LIN {X 0,Y 306.051,Z 523.216,A -85,B 0,C 180,E1 -15945.996,E2 -15945.996} C_VEL
LIN {X 0,Y 307.496,Z 515.084,A -85,B 0,C 180,E1 -15948.317,E2 -15948.317} C_VEL
LIN {X 0,Y 309.447,Z 505.284,A -85,B 0,C 180,E1 -15950.612,E2 -15950.612} C_VEL
LIN {X 0,Y 311.307,Z 495.226,A -85,B 0,C 180,E1 -15952.569,E2 -15952.569} C_VEL
LIN {X 0,Y 313.603,Z 483.236,A -85,B 0,C 180,E1 -15954.494,E2 -15954.494} C_VEL
LIN {X 0,Y 315.881,Z 471.244,A -85,B 0,C 180,E1 -15956.067,E2 -15956.067} C_VEL
LIN {X 0,Y 318.15,Z 458.217,A -85,B 0,C 180,E1 -15957.46,E2 -15957.46} C_VEL
LIN {X 0,Y 320.166,Z 444.237,A -85,B 0,C 180,E1 -15958.665,E2 -15958.665} C_VEL
LIN {X 0,Y 321.912,Z 430.188,A -85,B 0,C 180,E1 -15959.601,E2 -15959.601} C_VEL
LIN {X 0,Y 323.462,Z 414.88,A -85,B 0,C 180,E1 -15960.342,E2 -15960.342} C_VEL
LIN {X 0,Y 324.422,Z 399.961,A -85,B 0,C 180,E1 -15960.828,E2 -15960.828} C_VEL
LIN {X 0,Y 328.381,Z 286.379,A -85,B 0,C 180,E1 -15963.418,E2 -15963.418} C_VEL
LIN {X 0,Y 325.576,Z 267.519,A -85,B 0,C 180,E1 -15964.227,E2 -15964.227} C_VEL
LIN {X 0,Y 318.104,Z 251.499,A -85,B 0,C 180,E1 -15965.539,E2 -15965.539} C_VEL
LIN {X 0,Y 314.882,Z 244.85,A -85,B 0,C 180,E1 -15966.17,E2 -15966.17} C_VEL
LIN {X 0,Y 311.866,Z 233.893,A -85,B 0,C 180,E1 -15969.123,E2 -15969.123} C_VEL
LIN {X 0,Y 308.13,Z 222.045,A -85,B 0,C 180,E1 -15972.644,E2 -15972.644} C_VEL
LIN {X 0,Y 305.421,Z 214.153,A -85,B 0,C 180,E1 -15975.272,E2 -15975.272} C_VEL
LIN {X 0,Y 305.439,Z 214.046,A -85,B 0,C 180,E1 -15978.143,E2 -15978.143} C_VEL
LIN {X 0,Y 305.466,Z 214.044,A -85,B 0,C 180,E1 -15981.596,E2 -15981.596} C_VEL
LIN {X 0,Y 305.461,Z 214.064,A -85,B 0,C 180,E1 -15984.887,E2 -15984.887} C_VEL
LIN {X 0,Y 305.45,Z 214.039,A -85,B 0,C 180,E1 -15988.355,E2 -15988.355} C_VEL
LIN {X 0,Y 305.519,Z 214.049,A -85,B 0,C 180,E1 -15991.114,E2 -15991.114} C_VEL
LIN {X 0,Y 305.564,Z 214.015,A -85,B 0,C 180,E1 -15994.088,E2 -15994.088} C_VEL
LIN {X 0,Y 305.499,Z 214.048,A -85,B 0,C 180,E1 -15998.403,E2 -15998.403} C_VEL
LIN {X 0,Y 305.589,Z 214.042,A -85,B 0,C 180,E1 -16001.218,E2 -16001.218} C_VEL
LIN {X 0,Y 305.647,Z 214.031,A -85,B 0,C 180,E1 -16005.349,E2 -16005.349} C_VEL
LIN {X 0,Y 305.634,Z 214.033,A -85,B 0,C 180,E1 -16009.4,E2 -16009.4} C_VEL
LIN {X 0,Y 305.796,Z 214.021,A -85,B 0,C 180,E1 -16012.074,E2 -16012.074} C_VEL
LIN {X 0,Y 305.685,Z 214.021,A -85,B 0,C 180,E1 -16014.724,E2 -16014.724} C_VEL
LIN {X 0,Y 305.956,Z 213.986,A -85,B 0,C 180,E1 -16018.684,E2 -16018.684} C_VEL
LIN {X 0,Y 305.954,Z 214.001,A -85,B 0,C 180,E1 -16021.316,E2 -16021.316} C_VEL
LIN {X 0,Y 305.849,Z 214.007,A -85,B 0,C 180,E1 -16026.617,E2 -16026.617} C_VEL
LIN {X 0,Y 305.735,Z 214.025,A -85,B 0,C 180,E1 -16029.26,E2 -16029.26} C_VEL
LIN {X 0,Y 305.588,Z 214.042,A -85,B 0,C 180,E1 -16033.296,E2 -16033.296} C_VEL
LIN {X 0,Y 305.593,Z 214.033,A -85,B 0,C 180,E1 -16036.02,E2 -16036.02} C_VEL
LIN {X 0,Y 305.577,Z 214.037,A -85,B 0,C 180,E1 -16039.445,E2 -16039.445} C_VEL
LIN {X 0,Y 305.49,Z 214.051,A -85,B 0,C 180,E1 -16043.041,E2 -16043.041} C_VEL
LIN {X 0,Y 305.547,Z 214.047,A -85,B 0,C 180,E1 -16046.227,E2 -16046.227} C_VEL
LIN {X 0,Y 305.487,Z 214.024,A -85,B 0,C 180,E1 -16049.047,E2 -16049.047} C_VEL
LIN {X 0,Y 305.443,Z 214.064,A -85,B 0,C 180,E1 -16051.953,E2 -16051.953} C_VEL
LIN {X 0,Y 305.462,Z 214.034,A -85,B 0,C 180,E1 -16055.114,E2 -16055.114} C_VEL
LIN {X 0,Y 305.467,Z 214.048,A -85,B 0,C 180,E1 -16058.533,E2 -16058.533} C_VEL
LIN {X 0,Y 305.455,Z 214.059,A -85,B 0,C 180,E1 -16062.586,E2 -16062.586} C_VEL
LIN {X 0,Y 305.44,Z 214.214,A -85,B 0,C 180,E1 -16067.071,E2 -16067.071} C_VEL
LIN {X 0,Y 308.758,Z 224.691,A -85,B 0,C 180,E1 -16070.707,E2 -16070.707} C_VEL
LIN {X 0,Y 311.935,Z 235.816,A -85,B 0,C 180,E1 -16074.203,E2 -16074.203} C_VEL
LIN {X 0,Y 314.182,Z 244.627,A -85,B 0,C 180,E1 -16076.729,E2 -16076.729} C_VEL
LIN {X 0,Y 323.172,Z 263.666,A -85,B 0,C 180,E1 -16078.334,E2 -16078.334} C_VEL
LIN {X 0,Y 327.852,Z 288.604,A -85,B 0,C 180,E1 -16079.474,E2 -16079.474} C_VEL
LIN {X 0,Y 324.938,Z 389.323,A -85,B 0,C 180,E1 -16081.586,E2 -16081.586} C_VEL
LIN {X 0,Y 323.983,Z 403.831,A -85,B 0,C 180,E1 -16082.112,E2 -16082.112} C_VEL
LIN {X 0,Y 322.707,Z 417.842,A -85,B 0,C 180,E1 -16082.88,E2 -16082.88} C_VEL
LIN {X 0,Y 320.966,Z 431.274,A -85,B 0,C 180,E1 -16083.865,E2 -16083.865} C_VEL
LIN {X 0,Y 319.149,Z 444.305,A -85,B 0,C 180,E1 -16085.122,E2 -16085.122} C_VEL
LIN {X 0,Y 316.76,Z 456.973,A -85,B 0,C 180,E1 -16086.634,E2 -16086.634} C_VEL
LIN {X 0,Y 314.827,Z 466.573,A -85,B 0,C 180,E1 -16088.042,E2 -16088.042} C_VEL
LIN {X 0,Y 312.58,Z 477.226,A -85,B 0,C 180,E1 -16089.947,E2 -16089.947} C_VEL
LIN {X 0,Y 310.566,Z 486.129,A -85,B 0,C 180,E1 -16091.888,E2 -16091.888} C_VEL
LIN {X 0,Y 309.055,Z 493.449,A -85,B 0,C 180,E1 -16093.825,E2 -16093.825} C_VEL
LIN {X 0,Y 307.268,Z 500.557,A -85,B 0,C 180,E1 -16096.104,E2 -16096.104} C_VEL
LIN {X 0,Y 305.875,Z 506.971,A -85,B 0,C 180,E1 -16098.737,E2 -16098.737} C_VEL
LIN {X 0,Y 304.905,Z 511.827,A -85,B 0,C 180,E1 -16101.383,E2 -16101.383} C_VEL
LIN {X 0,Y 304.442,Z 514.574,A -85,B 0,C 180,E1 -16103.371,E2 -16103.371} C_VEL
LIN {X 0,Y 303.993,Z 517.05,A -85,B 0,C 180,E1 -16106.023,E2 -16106.023} C_VEL
LIN {X 0,Y 303.785,Z 518.285,A -85,B 0,C 180,E1 -16108.674,E2 -16108.674} C_VEL
LIN {X 0,Y 303.779,Z 518.309,A -85,B 0,C 180,E1 -16111.325,E2 -16111.325} C_VEL
LIN {X 0,Y 303.983,Z 517.128,A -85,B 0,C 180,E1 -16113.977,E2 -16113.977} C_VEL
LIN {X 0,Y 304.417,Z 514.706,A -85,B 0,C 180,E1 -16116.628,E2 -16116.628} C_VEL
LIN {X 0,Y 305.05,Z 510.973,A -85,B 0,C 180,E1 -16119.28,E2 -16119.28} C_VEL
LIN {X 0,Y 306.141,Z 505.797,A -85,B 0,C 180,E1 -16121.923,E2 -16121.923} C_VEL
LIN {X 0,Y 307.602,Z 499,A -85,B 0,C 180,E1 -16124.555,E2 -16124.555} C_VEL
LIN {X 0,Y 309.482,Z 491.522,A -85,B 0,C 180,E1 -16126.83,E2 -16126.83} C_VEL
LIN {X 0,Y 311.127,Z 483.786,A -85,B 0,C 180,E1 -16128.777,E2 -16128.777} C_VEL
LIN {X 0,Y 313.253,Z 474.492,A -85,B 0,C 180,E1 -16130.692,E2 -16130.692} C_VEL
LIN {X 0,Y 315.592,Z 463.192,A -85,B 0,C 180,E1 -16132.59,E2 -16132.59} C_VEL
LIN {X 0,Y 317.844,Z 451.718,A -85,B 0,C 180,E1 -16134.145,E2 -16134.145} C_VEL
LIN {X 0,Y 319.889,Z 439.506,A -85,B 0,C 180,E1 -16135.488,E2 -16135.488} C_VEL
LIN {X 0,Y 321.664,Z 426.703,A -85,B 0,C 180,E1 -16136.608,E2 -16136.608} C_VEL
LIN {X 0,Y 323.212,Z 413.053,A -85,B 0,C 180,E1 -16137.52,E2 -16137.52} C_VEL
LIN {X 0,Y 324.425,Z 398.92,A -85,B 0,C 180,E1 -16138.197,E2 -16138.197} C_VEL
LIN {X 0,Y 325.109,Z 385.652,A -85,B 0,C 180,E1 -16138.617,E2 -16138.617} C_VEL
LIN {X 0,Y 327.944,Z 288.805,A -85,B 0,C 180,E1 -16140.629,E2 -16140.629} C_VEL
LIN {X 0,Y 324.369,Z 269.366,A -85,B 0,C 180,E1 -16141.504,E2 -16141.504} C_VEL
LIN {X 0,Y 322.955,Z 263.152,A -85,B 0,C 180,E1 -16141.822,E2 -16141.822} C_VEL
LIN {X 0,Y 318.247,Z 253.023,A -85,B 0,C 180,E1 -16142.64,E2 -16142.64} C_VEL
LIN {X 0,Y 315.072,Z 249.483,A -85,B 0,C 180,E1 -16143.123,E2 -16143.123} C_VEL
LIN {X 0,Y 309.598,Z 245.583,A -85,B 0,C 180,E1 -16143.988,E2 -16143.988} C_VEL
LIN {X 0,Y 306.921,Z 243.119,A -85,B 0,C 180,E1 -16144.717,E2 -16144.717} C_VEL
LIN {X 0,Y 306.277,Z 241.768,A -85,B 0,C 180,E1 -16145.126,E2 -16145.126} C_VEL
LIN {X 0,Y 303.724,Z 232.189,A -85,B 0,C 180,E1 -16148.118,E2 -16148.118} C_VEL
LIN {X 0,Y 300.595,Z 222.006,A -85,B 0,C 180,E1 -16151.567,E2 -16151.567} C_VEL
LIN {X 0,Y 298.372,Z 214.997,A -85,B 0,C 180,E1 -16154.198,E2 -16154.198} C_VEL
LIN {X 0,Y 298.4,Z 214.929,A -85,B 0,C 180,E1 -16156.92,E2 -16156.92} C_VEL
LIN {X 0,Y 298.411,Z 214.921,A -85,B 0,C 180,E1 -16161.003,E2 -16161.003} C_VEL
LIN {X 0,Y 298.427,Z 214.922,A -85,B 0,C 180,E1 -16163.931,E2 -16163.931} C_VEL
LIN {X 0,Y 298.393,Z 214.942,A -85,B 0,C 180,E1 -16167.982,E2 -16167.982} C_VEL
LIN {X 0,Y 298.459,Z 214.9,A -85,B 0,C 180,E1 -16171.904,E2 -16171.904} C_VEL
LIN {X 0,Y 298.481,Z 214.931,A -85,B 0,C 180,E1 -16174.923,E2 -16174.923} C_VEL
LIN {X 0,Y 298.454,Z 214.926,A -85,B 0,C 180,E1 -16179.315,E2 -16179.315} C_VEL
LIN {X 0,Y 298.533,Z 214.924,A -85,B 0,C 180,E1 -16182.179,E2 -16182.179} C_VEL
LIN {X 0,Y 298.588,Z 214.91,A -85,B 0,C 180,E1 -16184.994,E2 -16184.994} C_VEL
LIN {X 0,Y 298.588,Z 214.911,A -85,B 0,C 180,E1 -16189.146,E2 -16189.146} C_VEL
LIN {X 0,Y 298.752,Z 214.887,A -85,B 0,C 180,E1 -16191.886,E2 -16191.886} C_VEL
LIN {X 0,Y 298.654,Z 214.911,A -85,B 0,C 180,E1 -16194.599,E2 -16194.599} C_VEL
LIN {X 0,Y 298.917,Z 214.876,A -85,B 0,C 180,E1 -16198.653,E2 -16198.653} C_VEL
LIN {X 0,Y 298.918,Z 214.863,A -85,B 0,C 180,E1 -16201.347,E2 -16201.347} C_VEL
LIN {X 0,Y 298.791,Z 214.888,A -85,B 0,C 180,E1 -16206.754,E2 -16206.754} C_VEL
LIN {X 0,Y 298.674,Z 214.896,A -85,B 0,C 180,E1 -16209.48,E2 -16209.48} C_VEL
LIN {X 0,Y 298.545,Z 214.912,A -85,B 0,C 180,E1 -16213.615,E2 -16213.615} C_VEL
LIN {X 0,Y 298.542,Z 214.919,A -85,B 0,C 180,E1 -16216.409,E2 -16216.409} C_VEL
LIN {X 0,Y 298.506,Z 214.927,A -85,B 0,C 180,E1 -16219.655,E2 -16219.655} C_VEL
LIN {X 0,Y 298.452,Z 214.934,A -85,B 0,C 180,E1 -16223.598,E2 -16223.598} C_VEL
LIN {X 0,Y 298.478,Z 214.895,A -85,B 0,C 180,E1 -16226.575,E2 -16226.575} C_VEL
LIN {X 0,Y 298.415,Z 214.941,A -85,B 0,C 180,E1 -16229.641,E2 -16229.641} C_VEL
LIN {X 0,Y 298.39,Z 214.913,A -85,B 0,C 180,E1 -16232.801,E2 -16232.801} C_VEL
LIN {X 0,Y 298.439,Z 214.917,A -85,B 0,C 180,E1 -16236.808,E2 -16236.808} C_VEL
LIN {X 0,Y 298.382,Z 214.928,A -85,B 0,C 180,E1 -16241.088,E2 -16241.088} C_VEL
LIN {X 0,Y 298.406,Z 215.139,A -85,B 0,C 180,E1 -16243.687,E2 -16243.687} C_VEL
LIN {X 0,Y 302.396,Z 226.886,A -85,B 0,C 180,E1 -16247.626,E2 -16247.626} C_VEL
LIN {X 0,Y 305.735,Z 237.627,A -85,B 0,C 180,E1 -16250.878,E2 -16250.878} C_VEL
LIN {X 0,Y 307.813,Z 245.088,A -85,B 0,C 180,E1 -16252.91,E2 -16252.91} C_VEL
LIN {X 0,Y 317.262,Z 264.383,A -85,B 0,C 180,E1 -16254.683,E2 -16254.683} C_VEL
LIN {X 0,Y 320.012,Z 270.972,A -85,B 0,C 180,E1 -16255.193,E2 -16255.193} C_VEL
LIN {X 0,Y 322.423,Z 287.669,A -85,B 0,C 180,E1 -16255.925,E2 -16255.925} C_VEL
LIN {X 0,Y 318.168,Z 404.092,A -85,B 0,C 180,E1 -16258.637,E2 -16258.637} C_VEL
LIN {X 0,Y 316.869,Z 419.944,A -85,B 0,C 180,E1 -16259.236,E2 -16259.236} C_VEL
LIN {X 0,Y 315.173,Z 434.989,A -85,B 0,C 180,E1 -16260.071,E2 -16260.071} C_VEL
LIN {X 0,Y 313.092,Z 449.727,A -85,B 0,C 180,E1 -16261.171,E2 -16261.171} C_VEL
LIN {X 0,Y 311.039,Z 462.669,A -85,B 0,C 180,E1 -16262.407,E2 -16262.407} C_VEL
LIN {X 0,Y 308.791,Z 474.892,A -85,B 0,C 180,E1 -16263.835,E2 -16263.835} C_VEL
LIN {X 0,Y 306.475,Z 486.249,A -85,B 0,C 180,E1 -16265.441,E2 -16265.441} C_VEL
LIN {X 0,Y 304.11,Z 498,A -85,B 0,C 180,E1 -16267.468,E2 -16267.468} C_VEL
LIN {X 0,Y 302.156,Z 508.06,A -85,B 0,C 180,E1 -16269.581,E2 -16269.581} C_VEL
LIN {X 0,Y 300.216,Z 517.34,A -85,B 0,C 180,E1 -16271.931,E2 -16271.931} C_VEL
LIN {X 0,Y 298.723,Z 525.226,A -85,B 0,C 180,E1 -16274.373,E2 -16274.373} C_VEL
LIN {X 0,Y 297.623,Z 532.156,A -85,B 0,C 180,E1 -16277.037,E2 -16277.037} C_VEL
LIN {X 0,Y 296.894,Z 537.721,A -85,B 0,C 180,E1 -16279.774,E2 -16279.774} C_VEL
LIN {X 0,Y 296.666,Z 540.935,A -85,B 0,C 180,E1 -16281.829,E2 -16281.829} C_VEL
LIN {X 0,Y 296.599,Z 544.1,A -85,B 0,C 180,E1 -16284.562,E2 -16284.562} C_VEL
LIN {X 0,Y 296.593,Z 545.984,A -85,B 0,C 180,E1 -16287.284,E2 -16287.284} C_VEL
LIN {X 0,Y 296.665,Z 546.621,A -85,B 0,C 180,E1 -16290.001,E2 -16290.001} C_VEL
LIN {X 0,Y 296.601,Z 545.974,A -85,B 0,C 180,E1 -16292.717,E2 -16292.717} C_VEL
LIN {X 0,Y 296.629,Z 543.871,A -85,B 0,C 180,E1 -16295.676,E2 -16295.676} C_VEL
LIN {X 0,Y 296.746,Z 539.931,A -85,B 0,C 180,E1 -16298.856,E2 -16298.856} C_VEL
LIN {X 0,Y 297.214,Z 535.079,A -85,B 0,C 180,E1 -16301.595,E2 -16301.595} C_VEL
LIN {X 0,Y 298.156,Z 528.731,A -85,B 0,C 180,E1 -16304.33,E2 -16304.33} C_VEL
LIN {X 0,Y 299.344,Z 521.826,A -85,B 0,C 180,E1 -16306.715,E2 -16306.715} C_VEL
LIN {X 0,Y 300.898,Z 513.46,A -85,B 0,C 180,E1 -16309.087,E2 -16309.087} C_VEL
LIN {X 0,Y 302.717,Z 504.915,A -85,B 0,C 180,E1 -16311.091,E2 -16311.091} C_VEL
LIN {X 0,Y 304.656,Z 494.842,A -85,B 0,C 180,E1 -16313.09,E2 -16313.09} C_VEL
LIN {X 0,Y 307.106,Z 482.838,A -85,B 0,C 180,E1 -16315.047,E2 -16315.047} C_VEL
LIN {X 0,Y 309.468,Z 470.819,A -85,B 0,C 180,E1 -16316.649,E2 -16316.649} C_VEL
LIN {X 0,Y 311.822,Z 457.755,A -85,B 0,C 180,E1 -16318.066,E2 -16318.066} C_VEL
LIN {X 0,Y 313.873,Z 444.099,A -85,B 0,C 180,E1 -16319.26,E2 -16319.26} C_VEL
LIN {X 0,Y 315.734,Z 429.579,A -85,B 0,C 180,E1 -16320.24,E2 -16320.24} C_VEL
LIN {X 0,Y 317.264,Z 415.014,A -85,B 0,C 180,E1 -16320.953,E2 -16320.953} C_VEL
LIN {X 0,Y 318.256,Z 400.286,A -85,B 0,C 180,E1 -16321.447,E2 -16321.447} C_VEL
LIN {X 0,Y 322.365,Z 287.404,A -85,B 0,C 180,E1 -16324.06,E2 -16324.06} C_VEL
LIN {X 0,Y 319.811,Z 270.111,A -85,B 0,C 180,E1 -16324.824,E2 -16324.824} C_VEL
LIN {X 0,Y 311.443,Z 252.373,A -85,B 0,C 180,E1 -16326.346,E2 -16326.346} C_VEL
LIN {X 0,Y 307.697,Z 244.879,A -85,B 0,C 180,E1 -16327.095,E2 -16327.095} C_VEL
LIN {X 0,Y 304.431,Z 233.257,A -85,B 0,C 180,E1 -16330.375,E2 -16330.375} C_VEL
LIN {X 0,Y 301.03,Z 222.831,A -85,B 0,C 180,E1 -16333.636,E2 -16333.636} C_VEL
LIN {X 0,Y 298.41,Z 215.032,A -85,B 0,C 180,E1 -16336.343,E2 -16336.343} C_VEL
LIN {X 0,Y 298.4,Z 214.939,A -85,B 0,C 180,E1 -16340.513,E2 -16340.513} C_VEL
LIN {X 0,Y 298.417,Z 214.932,A -85,B 0,C 180,E1 -16343.93,E2 -16343.93} C_VEL
LIN {X 0,Y 298.393,Z 214.914,A -85,B 0,C 180,E1 -16347.984,E2 -16347.984} C_VEL
LIN {X 0,Y 298.452,Z 214.912,A -85,B 0,C 180,E1 -16351.903,E2 -16351.903} C_VEL
LIN {X 0,Y 298.482,Z 214.907,A -85,B 0,C 180,E1 -16354.924,E2 -16354.924} C_VEL
LIN {X 0,Y 298.449,Z 214.929,A -85,B 0,C 180,E1 -16359.315,E2 -16359.315} C_VEL
LIN {X 0,Y 298.536,Z 214.914,A -85,B 0,C 180,E1 -16362.18,E2 -16362.18} C_VEL
LIN {X 0,Y 298.592,Z 214.914,A -85,B 0,C 180,E1 -16364.995,E2 -16364.995} C_VEL
LIN {X 0,Y 298.59,Z 214.913,A -85,B 0,C 180,E1 -16369.147,E2 -16369.147} C_VEL
LIN {X 0,Y 298.74,Z 214.897,A -85,B 0,C 180,E1 -16371.886,E2 -16371.886} C_VEL
LIN {X 0,Y 298.656,Z 214.896,A -85,B 0,C 180,E1 -16374.599,E2 -16374.599} C_VEL
LIN {X 0,Y 298.922,Z 214.862,A -85,B 0,C 180,E1 -16378.653,E2 -16378.653} C_VEL
LIN {X 0,Y 298.92,Z 214.877,A -85,B 0,C 180,E1 -16381.347,E2 -16381.347} C_VEL
LIN {X 0,Y 298.796,Z 214.884,A -85,B 0,C 180,E1 -16386.754,E2 -16386.754} C_VEL
LIN {X 0,Y 298.68,Z 214.906,A -85,B 0,C 180,E1 -16389.481,E2 -16389.481} C_VEL
LIN {X 0,Y 298.551,Z 214.922,A -85,B 0,C 180,E1 -16393.616,E2 -16393.616} C_VEL
LIN {X 0,Y 298.548,Z 214.911,A -85,B 0,C 180,E1 -16396.409,E2 -16396.409} C_VEL
LIN {X 0,Y 298.511,Z 214.916,A -85,B 0,C 180,E1 -16399.655,E2 -16399.655} C_VEL
LIN {X 0,Y 298.457,Z 214.924,A -85,B 0,C 180,E1 -16403.598,E2 -16403.598} C_VEL
LIN {X 0,Y 298.489,Z 214.919,A -85,B 0,C 180,E1 -16406.575,E2 -16406.575} C_VEL
LIN {X 0,Y 298.416,Z 214.908,A -85,B 0,C 180,E1 -16409.642,E2 -16409.642} C_VEL
LIN {X 0,Y 298.395,Z 214.934,A -85,B 0,C 180,E1 -16412.801,E2 -16412.801} C_VEL
LIN {X 0,Y 298.464,Z 214.927,A -85,B 0,C 180,E1 -16416.812,E2 -16416.812} C_VEL
LIN {X 0,Y 298.387,Z 214.928,A -85,B 0,C 180,E1 -16421.088,E2 -16421.088} C_VEL
LIN {X 0,Y 298.4,Z 214.929,A -85,B 0,C 180,E1 -16423.104,E2 -16423.104} C_VEL
LIN {X 0,Y 298.405,Z 215.112,A -85,B 0,C 180,E1 -16426.038,E2 -16426.038} C_VEL
LIN {X 0,Y 302.065,Z 226.571,A -85,B 0,C 180,E1 -16430.157,E2 -16430.157} C_VEL
LIN {X 0,Y 305.19,Z 237.535,A -85,B 0,C 180,E1 -16433.706,E2 -16433.706} C_VEL
LIN {X 0,Y 307.026,Z 244.659,A -85,B 0,C 180,E1 -16435.801,E2 -16435.801} C_VEL
LIN {X 0,Y 315.775,Z 262.591,A -85,B 0,C 180,E1 -16437.426,E2 -16437.426} C_VEL
LIN {X 0,Y 317.735,Z 267.319,A -85,B 0,C 180,E1 -16437.785,E2 -16437.785} C_VEL
LIN {X 0,Y 321.805,Z 289.209,A -85,B 0,C 180,E1 -16438.814,E2 -16438.814} C_VEL
LIN {X 0,Y 318.753,Z 390.353,A -85,B 0,C 180,E1 -16440.983,E2 -16440.983} C_VEL
LIN {X 0,Y 317.673,Z 405.29,A -85,B 0,C 180,E1 -16441.553,E2 -16441.553} C_VEL
LIN {X 0,Y 316.426,Z 418.4,A -85,B 0,C 180,E1 -16442.296,E2 -16442.296} C_VEL
LIN {X 0,Y 314.534,Z 432.372,A -85,B 0,C 180,E1 -16443.351,E2 -16443.351} C_VEL
LIN {X 0,Y 312.513,Z 445.92,A -85,B 0,C 180,E1 -16444.704,E2 -16444.704} C_VEL
LIN {X 0,Y 310.262,Z 457.38,A -85,B 0,C 180,E1 -16446.115,E2 -16446.115} C_VEL
LIN {X 0,Y 308.259,Z 466.956,A -85,B 0,C 180,E1 -16447.549,E2 -16447.549} C_VEL
LIN {X 0,Y 305.912,Z 477.594,A -85,B 0,C 180,E1 -16449.491,E2 -16449.491} C_VEL
LIN {X 0,Y 303.73,Z 486.873,A -85,B 0,C 180,E1 -16451.568,E2 -16451.568} C_VEL
LIN {X 0,Y 301.938,Z 494.885,A -85,B 0,C 180,E1 -16453.78,E2 -16453.78} C_VEL
LIN {X 0,Y 300.381,Z 500.899,A -85,B 0,C 180,E1 -16455.778,E2 -16455.778} C_VEL
LIN {X 0,Y 298.905,Z 507.311,A -85,B 0,C 180,E1 -16458.471,E2 -16458.471} C_VEL
LIN {X 0,Y 297.894,Z 512.164,A -85,B 0,C 180,E1 -16461.179,E2 -16461.179} C_VEL
LIN {X 0,Y 297.39,Z 514.909,A -85,B 0,C 180,E1 -16463.214,E2 -16463.214} C_VEL
LIN {X 0,Y 296.931,Z 517.383,A -85,B 0,C 180,E1 -16465.928,E2 -16465.928} C_VEL
LIN {X 0,Y 296.697,Z 518.618,A -85,B 0,C 180,E1 -16468.642,E2 -16468.642} C_VEL
LIN {X 0,Y 296.691,Z 518.642,A -85,B 0,C 180,E1 -16471.357,E2 -16471.357} C_VEL
LIN {X 0,Y 296.921,Z 517.46,A -85,B 0,C 180,E1 -16474.071,E2 -16474.071} C_VEL
LIN {X 0,Y 297.369,Z 515.039,A -85,B 0,C 180,E1 -16476.786,E2 -16476.786} C_VEL
LIN {X 0,Y 298.05,Z 511.308,A -85,B 0,C 180,E1 -16479.5,E2 -16479.5} C_VEL
LIN {X 0,Y 299.192,Z 506.136,A -85,B 0,C 180,E1 -16482.204,E2 -16482.204} C_VEL
LIN {X 0,Y 300.737,Z 499.342,A -85,B 0,C 180,E1 -16484.895,E2 -16484.895} C_VEL
LIN {X 0,Y 302.682,Z 491.871,A -85,B 0,C 180,E1 -16487.219,E2 -16487.219} C_VEL
LIN {X 0,Y 304.404,Z 484.144,A -85,B 0,C 180,E1 -16489.207,E2 -16489.207} C_VEL
LIN {X 0,Y 306.639,Z 474.861,A -85,B 0,C 180,E1 -16491.16,E2 -16491.16} C_VEL
LIN {X 0,Y 309.075,Z 463.578,A -85,B 0,C 180,E1 -16493.093,E2 -16493.093} C_VEL
LIN {X 0,Y 311.395,Z 452.129,A -85,B 0,C 180,E1 -16494.678,E2 -16494.678} C_VEL
LIN {X 0,Y 313.639,Z 439.181,A -85,B 0,C 180,E1 -16496.121,E2 -16496.121} C_VEL
LIN {X 0,Y 315.367,Z 427.204,A -85,B 0,C 180,E1 -16497.182,E2 -16497.182} C_VEL
LIN {X 0,Y 316.975,Z 413.646,A -85,B 0,C 180,E1 -16498.108,E2 -16498.108} C_VEL
LIN {X 0,Y 318.218,Z 399.681,A -85,B 0,C 180,E1 -16498.798,E2 -16498.798} C_VEL
LIN {X 0,Y 319.005,Z 385.246,A -85,B 0,C 180,E1 -16499.262,E2 -16499.262} C_VEL
LIN {X 0,Y 321.873,Z 289.056,A -85,B 0,C 180,E1 -16501.301,E2 -16501.301} C_VEL
LIN {X 0,Y 317.455,Z 266.356,A -85,B 0,C 180,E1 -16502.393,E2 -16502.393} C_VEL
LIN {X 0,Y 308.804,Z 248.284,A -85,B 0,C 180,E1 -16503.961,E2 -16503.961} C_VEL
LIN {X 0,Y 306.963,Z 244.446,A -85,B 0,C 180,E1 -16504.36,E2 -16504.36} C_VEL
LIN {X 0,Y 306.277,Z 241.768,A -85,B 0,C 180,E1 -16505.126,E2 -16505.126} C_VEL
LIN {X 0,Y 304.938,Z 238.984,A -85,B 0,C 180,E1 -16506.067,E2 -16506.067} C_VEL
LIN {X 0,Y 301.039,Z 235.343,A -85,B 0,C 180,E1 -16507.649,E2 -16507.649} C_VEL
LIN {X 0,Y 297.75,Z 232.605,A -85,B 0,C 180,E1 -16508.947,E2 -16508.947} C_VEL
LIN {X 0,Y 295.968,Z 230.198,A -85,B 0,C 180,E1 -16509.945,E2 -16509.945} C_VEL
LIN {X 0,Y 295.61,Z 229.274,A -85,B 0,C 180,E1 -16510.28,E2 -16510.28} C_VEL
LIN {X 0,Y 292.195,Z 218.489,A -85,B 0,C 180,E1 -16514.227,E2 -16514.227} C_VEL
LIN {X 0,Y 291.313,Z 215.876,A -85,B 0,C 180,E1 -16515.329,E2 -16515.329} C_VEL
LIN {X 0,Y 291.33,Z 215.804,A -85,B 0,C 180,E1 -16519.357,E2 -16519.357} C_VEL
LIN {X 0,Y 291.421,Z 215.812,A -85,B 0,C 180,E1 -16522.921,E2 -16522.921} C_VEL
LIN {X 0,Y 291.341,Z 215.797,A -85,B 0,C 180,E1 -16526.301,E2 -16526.301} C_VEL
LIN {X 0,Y 291.383,Z 215.785,A -85,B 0,C 180,E1 -16530.259,E2 -16530.259} C_VEL
LIN {X 0,Y 291.413,Z 215.81,A -85,B 0,C 180,E1 -16534.271,E2 -16534.271} C_VEL
LIN {X 0,Y 291.384,Z 215.809,A -85,B 0,C 180,E1 -16537.299,E2 -16537.299} C_VEL
LIN {X 0,Y 291.454,Z 215.795,A -85,B 0,C 180,E1 -16540.27,E2 -16540.27} C_VEL
LIN {X 0,Y 291.535,Z 215.786,A -85,B 0,C 180,E1 -16544.634,E2 -16544.634} C_VEL
LIN {X 0,Y 291.531,Z 215.787,A -85,B 0,C 180,E1 -16548.88,E2 -16548.88} C_VEL
LIN {X 0,Y 291.703,Z 215.766,A -85,B 0,C 180,E1 -16551.688,E2 -16551.688} C_VEL
LIN {X 0,Y 291.625,Z 215.785,A -85,B 0,C 180,E1 -16554.468,E2 -16554.468} C_VEL
LIN {X 0,Y 291.884,Z 215.752,A -85,B 0,C 180,E1 -16558.62,E2 -16558.62} C_VEL
LIN {X 0,Y 291.884,Z 215.739,A -85,B 0,C 180,E1 -16561.379,E2 -16561.379} C_VEL
LIN {X 0,Y 291.74,Z 215.768,A -85,B 0,C 180,E1 -16566.918,E2 -16566.918} C_VEL
LIN {X 0,Y 291.623,Z 215.773,A -85,B 0,C 180,E1 -16569.712,E2 -16569.712} C_VEL
LIN {X 0,Y 291.515,Z 215.787,A -85,B 0,C 180,E1 -16573.95,E2 -16573.95} C_VEL
LIN {X 0,Y 291.481,Z 215.797,A -85,B 0,C 180,E1 -16576.818,E2 -16576.818} C_VEL
LIN {X 0,Y 291.445,Z 215.807,A -85,B 0,C 180,E1 -16579.875,E2 -16579.875} C_VEL
LIN {X 0,Y 291.394,Z 215.807,A -85,B 0,C 180,E1 -16584.206,E2 -16584.206} C_VEL
LIN {X 0,Y 291.411,Z 215.778,A -85,B 0,C 180,E1 -16587.272,E2 -16587.272} C_VEL
LIN {X 0,Y 291.332,Z 215.815,A -85,B 0,C 180,E1 -16590.437,E2 -16590.437} C_VEL
LIN {X 0,Y 291.339,Z 215.798,A -85,B 0,C 180,E1 -16593.699,E2 -16593.699} C_VEL
LIN {X 0,Y 291.367,Z 215.794,A -85,B 0,C 180,E1 -16597.253,E2 -16597.253} C_VEL
LIN {X 0,Y 291.327,Z 215.812,A -85,B 0,C 180,E1 -16600.643,E2 -16600.643} C_VEL
LIN {X 0,Y 291.374,Z 216.033,A -85,B 0,C 180,E1 -16602.547,E2 -16602.547} C_VEL
LIN {X 0,Y 295.53,Z 228.279,A -85,B 0,C 180,E1 -16606.835,E2 -16606.835} C_VEL
LIN {X 0,Y 298.878,Z 238.898,A -85,B 0,C 180,E1 -16610.172,E2 -16610.172} C_VEL
LIN {X 0,Y 300.666,Z 245.172,A -85,B 0,C 180,E1 -16611.934,E2 -16611.934} C_VEL
LIN {X 0,Y 309.736,Z 263.232,A -85,B 0,C 180,E1 -16613.71,E2 -16613.71} C_VEL
LIN {X 0,Y 314.334,Z 273.671,A -85,B 0,C 180,E1 -16614.583,E2 -16614.583} C_VEL
LIN {X 0,Y 316.46,Z 288.587,A -85,B 0,C 180,E1 -16615.255,E2 -16615.255} C_VEL
LIN {X 0,Y 312.018,Z 404.386,A -85,B 0,C 180,E1 -16617.994,E2 -16617.994} C_VEL
LIN {X 0,Y 310.7,Z 420.044,A -85,B 0,C 180,E1 -16618.604,E2 -16618.604} C_VEL
LIN {X 0,Y 309.019,Z 434.446,A -85,B 0,C 180,E1 -16619.412,E2 -16619.412} C_VEL
LIN {X 0,Y 307.006,Z 448.333,A -85,B 0,C 180,E1 -16620.446,E2 -16620.446} C_VEL
LIN {X 0,Y 304.714,Z 462.237,A -85,B 0,C 180,E1 -16621.784,E2 -16621.784} C_VEL
LIN {X 0,Y 302.358,Z 474.485,A -85,B 0,C 180,E1 -16623.235,E2 -16623.235} C_VEL
LIN {X 0,Y 299.739,Z 486.893,A -85,B 0,C 180,E1 -16625.037,E2 -16625.037} C_VEL
LIN {X 0,Y 297.442,Z 497.778,A -85,B 0,C 180,E1 -16626.966,E2 -16626.966} C_VEL
LIN {X 0,Y 295.428,Z 507.698,A -85,B 0,C 180,E1 -16629.095,E2 -16629.095} C_VEL
LIN {X 0,Y 293.373,Z 516.986,A -85,B 0,C 180,E1 -16631.494,E2 -16631.494} C_VEL
LIN {X 0,Y 291.87,Z 524.672,A -85,B 0,C 180,E1 -16633.925,E2 -16633.925} C_VEL
LIN {X 0,Y 290.61,Z 531.812,A -85,B 0,C 180,E1 -16636.719,E2 -16636.719} C_VEL
LIN {X 0,Y 289.828,Z 537.381,A -85,B 0,C 180,E1 -16639.522,E2 -16639.522} C_VEL
LIN {X 0,Y 289.587,Z 540.598,A -85,B 0,C 180,E1 -16641.628,E2 -16641.628} C_VEL
LIN {X 0,Y 289.535,Z 543.767,A -85,B 0,C 180,E1 -16644.429,E2 -16644.429} C_VEL
LIN {X 0,Y 289.517,Z 545.652,A -85,B 0,C 180,E1 -16647.218,E2 -16647.218} C_VEL
LIN {X 0,Y 289.576,Z 546.289,A -85,B 0,C 180,E1 -16650.001,E2 -16650.001} C_VEL
LIN {X 0,Y 289.525,Z 545.641,A -85,B 0,C 180,E1 -16652.783,E2 -16652.783} C_VEL
LIN {X 0,Y 289.55,Z 543.683,A -85,B 0,C 180,E1 -16655.643,E2 -16655.643} C_VEL
LIN {X 0,Y 289.613,Z 540.566,A -85,B 0,C 180,E1 -16658.373,E2 -16658.373} C_VEL
LIN {X 0,Y 289.972,Z 536.049,A -85,B 0,C 180,E1 -16661.18,E2 -16661.18} C_VEL
LIN {X 0,Y 290.904,Z 530.087,A -85,B 0,C 180,E1 -16663.981,E2 -16663.981} C_VEL
LIN {X 0,Y 292.238,Z 522.513,A -85,B 0,C 180,E1 -16666.774,E2 -16666.774} C_VEL
LIN {X 0,Y 293.845,Z 514.366,A -85,B 0,C 180,E1 -16669.2,E2 -16669.2} C_VEL
LIN {X 0,Y 295.704,Z 506.067,A -85,B 0,C 180,E1 -16671.251,E2 -16671.251} C_VEL
LIN {X 0,Y 297.736,Z 496.02,A -85,B 0,C 180,E1 -16673.342,E2 -16673.342} C_VEL
LIN {X 0,Y 300.148,Z 484.607,A -85,B 0,C 180,E1 -16675.298,E2 -16675.298} C_VEL
LIN {X 0,Y 302.573,Z 473.007,A -85,B 0,C 180,E1 -16676.932,E2 -16676.932} C_VEL
LIN {X 0,Y 304.97,Z 460.481,A -85,B 0,C 180,E1 -16678.379,E2 -16678.379} C_VEL
LIN {X 0,Y 307.138,Z 447.071,A -85,B 0,C 180,E1 -16679.635,E2 -16679.635} C_VEL
LIN {X 0,Y 309.14,Z 432.857,A -85,B 0,C 180,E1 -16680.67,E2 -16680.67} C_VEL
LIN {X 0,Y 310.791,Z 418.761,A -85,B 0,C 180,E1 -16681.434,E2 -16681.434} C_VEL
LIN {X 0,Y 312.007,Z 403.529,A -85,B 0,C 180,E1 -16682.009,E2 -16682.009} C_VEL
LIN {X 0,Y 316.388,Z 288.477,A -85,B 0,C 180,E1 -16684.726,E2 -16684.726} C_VEL
LIN {X 0,Y 314.056,Z 272.698,A -85,B 0,C 180,E1 -16685.446,E2 -16685.446} C_VEL
LIN {X 0,Y 305.956,Z 255.613,A -85,B 0,C 180,E1 -16686.971,E2 -16686.971} C_VEL
LIN {X 0,Y 300.543,Z 244.815,A -85,B 0,C 180,E1 -16688.088,E2 -16688.088} C_VEL
LIN {X 0,Y 297.227,Z 233.459,A -85,B 0,C 180,E1 -16691.458,E2 -16691.458} C_VEL
LIN {X 0,Y 294.4,Z 224.866,A -85,B 0,C 180,E1 -16694.261,E2 -16694.261} C_VEL
LIN {X 0,Y 291.348,Z 215.928,A -85,B 0,C 180,E1 -16697.481,E2 -16697.481} C_VEL
LIN {X 0,Y 291.346,Z 215.806,A -85,B 0,C 180,E1 -16701.158,E2 -16701.158} C_VEL
LIN {X 0,Y 291.378,Z 215.818,A -85,B 0,C 180,E1 -16704.629,E2 -16704.629} C_VEL
LIN {X 0,Y 291.37,Z 215.788,A -85,B 0,C 180,E1 -16707.951,E2 -16707.951} C_VEL
LIN {X 0,Y 291.377,Z 215.807,A -85,B 0,C 180,E1 -16711.158,E2 -16711.158} C_VEL
LIN {X 0,Y 291.411,Z 215.778,A -85,B 0,C 180,E1 -16714.272,E2 -16714.272} C_VEL
LIN {X 0,Y 291.381,Z 215.814,A -85,B 0,C 180,E1 -16717.3,E2 -16717.3} C_VEL
LIN {X 0,Y 291.457,Z 215.807,A -85,B 0,C 180,E1 -16720.27,E2 -16720.27} C_VEL
LIN {X 0,Y 291.554,Z 215.791,A -85,B 0,C 180,E1 -16724.624,E2 -16724.624} C_VEL
LIN {X 0,Y 291.534,Z 215.794,A -85,B 0,C 180,E1 -16728.881,E2 -16728.881} C_VEL
LIN {X 0,Y 291.687,Z 215.773,A -85,B 0,C 180,E1 -16731.688,E2 -16731.688} C_VEL
LIN {X 0,Y 291.626,Z 215.771,A -85,B 0,C 180,E1 -16734.468,E2 -16734.468} C_VEL
LIN {X 0,Y 291.888,Z 215.738,A -85,B 0,C 180,E1 -16738.621,E2 -16738.621} C_VEL
LIN {X 0,Y 291.887,Z 215.752,A -85,B 0,C 180,E1 -16741.38,E2 -16741.38} C_VEL
LIN {X 0,Y 291.745,Z 215.76,A -85,B 0,C 180,E1 -16746.918,E2 -16746.918} C_VEL
LIN {X 0,Y 291.629,Z 215.785,A -85,B 0,C 180,E1 -16749.712,E2 -16749.712} C_VEL
LIN {X 0,Y 291.521,Z 215.797,A -85,B 0,C 180,E1 -16753.951,E2 -16753.951} C_VEL
LIN {X 0,Y 291.487,Z 215.793,A -85,B 0,C 180,E1 -16756.818,E2 -16756.818} C_VEL
LIN {X 0,Y 291.451,Z 215.795,A -85,B 0,C 180,E1 -16759.875,E2 -16759.875} C_VEL
LIN {X 0,Y 291.4,Z 215.805,A -85,B 0,C 180,E1 -16764.206,E2 -16764.206} C_VEL
LIN {X 0,Y 291.421,Z 215.787,A -85,B 0,C 180,E1 -16767.272,E2 -16767.272} C_VEL
LIN {X 0,Y 291.334,Z 215.801,A -85,B 0,C 180,E1 -16770.438,E2 -16770.438} C_VEL
LIN {X 0,Y 291.345,Z 215.797,A -85,B 0,C 180,E1 -16773.699,E2 -16773.699} C_VEL
LIN {X 0,Y 291.394,Z 215.814,A -85,B 0,C 180,E1 -16777.259,E2 -16777.259} C_VEL
LIN {X 0,Y 291.334,Z 215.801,A -85,B 0,C 180,E1 -16780.643,E2 -16780.643} C_VEL
LIN {X 0,Y 291.33,Z 215.981,A -85,B 0,C 180,E1 -16784.904,E2 -16784.904} C_VEL
LIN {X 0,Y 293.942,Z 224.001,A -85,B 0,C 180,E1 -16787.974,E2 -16787.974} C_VEL
LIN {X 0,Y 296.53,Z 232.385,A -85,B 0,C 180,E1 -16790.926,E2 -16790.926} C_VEL
LIN {X 0,Y 299.392,Z 242.945,A -85,B 0,C 180,E1 -16794.345,E2 -16794.345} C_VEL
LIN {X 0,Y 299.999,Z 244.96,A -85,B 0,C 180,E1 -16794.853,E2 -16794.853} C_VEL
LIN {X 0,Y 306.936,Z 258.72,A -85,B 0,C 180,E1 -16796.199,E2 -16796.199} C_VEL
LIN {X 0,Y 311.978,Z 269.509,A -85,B 0,C 180,E1 -16797.136,E2 -16797.136} C_VEL
LIN {X 0,Y 315.77,Z 289.864,A -85,B 0,C 180,E1 -16798.127,E2 -16798.127} C_VEL
LIN {X 0,Y 313.088,Z 378.403,A -85,B 0,C 180,E1 -16800.036,E2 -16800.036} C_VEL
LIN {X 0,Y 312.382,Z 394.807,A -85,B 0,C 180,E1 -16800.472,E2 -16800.472} C_VEL
LIN {X 0,Y 311.311,Z 408.277,A -85,B 0,C 180,E1 -16801.055,E2 -16801.055} C_VEL
LIN {X 0,Y 309.889,Z 421.439,A -85,B 0,C 180,E1 -16801.863,E2 -16801.863} C_VEL
LIN {X 0,Y 308.069,Z 433.887,A -85,B 0,C 180,E1 -16802.854,E2 -16802.854} C_VEL
LIN {X 0,Y 306.132,Z 446.355,A -85,B 0,C 180,E1 -16804.139,E2 -16804.139} C_VEL
LIN {X 0,Y 303.818,Z 457.782,A -85,B 0,C 180,E1 -16805.576,E2 -16805.576} C_VEL
LIN {X 0,Y 301.727,Z 467.338,A -85,B 0,C 180,E1 -16807.036,E2 -16807.036} C_VEL
LIN {X 0,Y 299.289,Z 477.96,A -85,B 0,C 180,E1 -16809.016,E2 -16809.016} C_VEL
LIN {X 0,Y 296.901,Z 487.626,A -85,B 0,C 180,E1 -16811.236,E2 -16811.236} C_VEL
LIN {X 0,Y 295.127,Z 495.234,A -85,B 0,C 180,E1 -16813.395,E2 -16813.395} C_VEL
LIN {X 0,Y 293.482,Z 501.243,A -85,B 0,C 180,E1 -16815.437,E2 -16815.437} C_VEL
LIN {X 0,Y 291.933,Z 507.651,A -85,B 0,C 180,E1 -16818.192,E2 -16818.192} C_VEL
LIN {X 0,Y 290.864,Z 512.501,A -85,B 0,C 180,E1 -16820.964,E2 -16820.964} C_VEL
LIN {X 0,Y 290.333,Z 515.244,A -85,B 0,C 180,E1 -16823.048,E2 -16823.048} C_VEL
LIN {X 0,Y 289.871,Z 517.716,A -85,B 0,C 180,E1 -16825.828,E2 -16825.828} C_VEL
LIN {X 0,Y 289.612,Z 518.95,A -85,B 0,C 180,E1 -16828.609,E2 -16828.609} C_VEL
LIN {X 0,Y 289.605,Z 518.974,A -85,B 0,C 180,E1 -16831.39,E2 -16831.39} C_VEL
LIN {X 0,Y 289.861,Z 517.791,A -85,B 0,C 180,E1 -16834.171,E2 -16834.171} C_VEL
LIN {X 0,Y 290.371,Z 515.219,A -85,B 0,C 180,E1 -16837.092,E2 -16837.092} C_VEL
LIN {X 0,Y 291.04,Z 511.643,A -85,B 0,C 180,E1 -16839.731,E2 -16839.731} C_VEL
LIN {X 0,Y 292.234,Z 506.475,A -85,B 0,C 180,E1 -16842.499,E2 -16842.499} C_VEL
LIN {X 0,Y 293.889,Z 499.684,A -85,B 0,C 180,E1 -16845.25,E2 -16845.25} C_VEL
LIN {X 0,Y 295.888,Z 492.22,A -85,B 0,C 180,E1 -16847.628,E2 -16847.628} C_VEL
LIN {X 0,Y 297.699,Z 484.502,A -85,B 0,C 180,E1 -16849.657,E2 -16849.657} C_VEL
LIN {X 0,Y 300.04,Z 475.229,A -85,B 0,C 180,E1 -16851.648,E2 -16851.648} C_VEL
LIN {X 0,Y 302.582,Z 463.963,A -85,B 0,C 180,E1 -16853.619,E2 -16853.619} C_VEL
LIN {X 0,Y 304.969,Z 452.539,A -85,B 0,C 180,E1 -16855.234,E2 -16855.234} C_VEL
LIN {X 0,Y 307.231,Z 440.063,A -85,B 0,C 180,E1 -16856.658,E2 -16856.658} C_VEL
LIN {X 0,Y 309.093,Z 427.698,A -85,B 0,C 180,E1 -16857.782,E2 -16857.782} C_VEL
LIN {X 0,Y 310.751,Z 414.239,A -85,B 0,C 180,E1 -16858.723,E2 -16858.723} C_VEL
LIN {X 0,Y 312.112,Z 399.513,A -85,B 0,C 180,E1 -16859.462,E2 -16859.462} C_VEL
LIN {X 0,Y 312.945,Z 384.841,A -85,B 0,C 180,E1 -16859.932,E2 -16859.932} C_VEL
LIN {X 0,Y 315.938,Z 291.066,A -85,B 0,C 180,E1 -16861.944,E2 -16861.944} C_VEL
LIN {X 0,Y 312.88,Z 273.847,A -85,B 0,C 180,E1 -16862.759,E2 -16862.759} C_VEL
LIN {X 0,Y 311.818,Z 269.209,A -85,B 0,C 180,E1 -16863.014,E2 -16863.014} C_VEL
LIN {X 0,Y 303.674,Z 252.124,A -85,B 0,C 180,E1 -16864.545,E2 -16864.545} C_VEL
LIN {X 0,Y 299.864,Z 244.639,A -85,B 0,C 180,E1 -16865.32,E2 -16865.32} C_VEL
LIN {X 0,Y 297.322,Z 235.05,A -85,B 0,C 180,E1 -16868.312,E2 -16868.312} C_VEL
LIN {X 0,Y 295.61,Z 229.274,A -85,B 0,C 180,E1 -16870.28,E2 -16870.28} C_VEL
LIN {X 0,Y 294.166,Z 226.786,A -85,B 0,C 180,E1 -16871.281,E2 -16871.281} C_VEL
LIN {X 0,Y 290.213,Z 223.721,A -85,B 0,C 180,E1 -16872.96,E2 -16872.96} C_VEL
LIN {X 0,Y 286.922,Z 221.431,A -85,B 0,C 180,E1 -16874.339,E2 -16874.339} C_VEL
LIN {X 0,Y 285.126,Z 219.337,A -85,B 0,C 180,E1 -16875.401,E2 -16875.401} C_VEL
LIN {X 0,Y 284.755,Z 218.508,A -85,B 0,C 180,E1 -16875.757,E2 -16875.757} C_VEL
LIN {X 0,Y 284.272,Z 216.764,A -85,B 0,C 180,E1 -16876.533,E2 -16876.533} C_VEL
LIN {X 0,Y 284.304,Z 216.675,A -85,B 0,C 180,E1 -16880.023,E2 -16880.023} C_VEL
LIN {X 0,Y 284.346,Z 216.679,A -85,B 0,C 180,E1 -16883.616,E2 -16883.616} C_VEL
LIN {X 0,Y 284.304,Z 216.686,A -85,B 0,C 180,E1 -16887.189,E2 -16887.189} C_VEL
LIN {X 0,Y 284.354,Z 216.658,A -85,B 0,C 180,E1 -16890.375,E2 -16890.375} C_VEL
LIN {X 0,Y 284.374,Z 216.677,A -85,B 0,C 180,E1 -16893.586,E2 -16893.586} C_VEL
LIN {X 0,Y 284.364,Z 216.679,A -85,B 0,C 180,E1 -16896.706,E2 -16896.706} C_VEL
LIN {X 0,Y 284.399,Z 216.68,A -85,B 0,C 180,E1 -16901.261,E2 -16901.261} C_VEL
LIN {X 0,Y 284.473,Z 216.664,A -85,B 0,C 180,E1 -16904.469,E2 -16904.469} C_VEL
LIN {X 0,Y 284.483,Z 216.663,A -85,B 0,C 180,E1 -16908.601,E2 -16908.601} C_VEL
LIN {X 0,Y 284.653,Z 216.646,A -85,B 0,C 180,E1 -16911.481,E2 -16911.481} C_VEL
LIN {X 0,Y 284.596,Z 216.66,A -85,B 0,C 180,E1 -16914.331,E2 -16914.331} C_VEL
LIN {X 0,Y 284.85,Z 216.627,A -85,B 0,C 180,E1 -16918.586,E2 -16918.586} C_VEL
LIN {X 0,Y 284.85,Z 216.615,A -85,B 0,C 180,E1 -16921.414,E2 -16921.414} C_VEL
LIN {X 0,Y 284.692,Z 216.647,A -85,B 0,C 180,E1 -16927.09,E2 -16927.09} C_VEL
LIN {X 0,Y 284.561,Z 216.653,A -85,B 0,C 180,E1 -16929.955,E2 -16929.955} C_VEL
LIN {X 0,Y 284.475,Z 216.664,A -85,B 0,C 180,E1 -16934.303,E2 -16934.303} C_VEL
LIN {X 0,Y 284.419,Z 216.673,A -85,B 0,C 180,E1 -16937.248,E2 -16937.248} C_VEL
LIN {X 0,Y 284.373,Z 216.684,A -85,B 0,C 180,E1 -16940.242,E2 -16940.242} C_VEL
LIN {X 0,Y 284.363,Z 216.685,A -85,B 0,C 180,E1 -16943.875,E2 -16943.875} C_VEL
LIN {X 0,Y 284.387,Z 216.651,A -85,B 0,C 180,E1 -16947.172,E2 -16947.172} C_VEL
LIN {X 0,Y 284.309,Z 216.695,A -85,B 0,C 180,E1 -16950.099,E2 -16950.099} C_VEL
LIN {X 0,Y 284.3,Z 216.667,A -85,B 0,C 180,E1 -16952.946,E2 -16952.946} C_VEL
LIN {X 0,Y 284.331,Z 216.677,A -85,B 0,C 180,E1 -16956.386,E2 -16956.386} C_VEL
LIN {X 0,Y 284.301,Z 216.698,A -85,B 0,C 180,E1 -16959.995,E2 -16959.995} C_VEL
LIN {X 0,Y 284.331,Z 216.963,A -85,B 0,C 180,E1 -16961.332,E2 -16961.332} C_VEL
LIN {X 0,Y 287.778,Z 227.06,A -85,B 0,C 180,E1 -16965.09,E2 -16965.09} C_VEL
LIN {X 0,Y 290.661,Z 235.749,A -85,B 0,C 180,E1 -16968.031,E2 -16968.031} C_VEL
LIN {X 0,Y 293.411,Z 244.981,A -85,B 0,C 180,E1 -16970.857,E2 -16970.857} C_VEL
LIN {X 0,Y 302.147,Z 261.967,A -85,B 0,C 180,E1 -16972.664,E2 -16972.664} C_VEL
LIN {X 0,Y 308.594,Z 275.961,A -85,B 0,C 180,E1 -16973.927,E2 -16973.927} C_VEL
LIN {X 0,Y 310.528,Z 289.688,A -85,B 0,C 180,E1 -16974.564,E2 -16974.564} C_VEL
LIN {X 0,Y 306.034,Z 403.379,A -85,B 0,C 180,E1 -16977.291,E2 -16977.291} C_VEL
LIN {X 0,Y 304.731,Z 418.576,A -85,B 0,C 180,E1 -16977.868,E2 -16977.868} C_VEL
LIN {X 0,Y 302.895,Z 433.903,A -85,B 0,C 180,E1 -16978.725,E2 -16978.725} C_VEL
LIN {X 0,Y 300.714,Z 448.5,A -85,B 0,C 180,E1 -16979.834,E2 -16979.834} C_VEL
LIN {X 0,Y 298.43,Z 461.806,A -85,B 0,C 180,E1 -16981.134,E2 -16981.134} C_VEL
LIN {X 0,Y 295.978,Z 474.078,A -85,B 0,C 180,E1 -16982.61,E2 -16982.61} C_VEL
LIN {X 0,Y 293.193,Z 486.507,A -85,B 0,C 180,E1 -16984.44,E2 -16984.44} C_VEL
LIN {X 0,Y 290.686,Z 498.12,A -85,B 0,C 180,E1 -16986.56,E2 -16986.56} C_VEL
LIN {X 0,Y 288.732,Z 507.337,A -85,B 0,C 180,E1 -16988.586,E2 -16988.586} C_VEL
LIN {X 0,Y 286.54,Z 516.632,A -85,B 0,C 180,E1 -16991.036,E2 -16991.036} C_VEL
LIN {X 0,Y 284.956,Z 524.324,A -85,B 0,C 180,E1 -16993.524,E2 -16993.524} C_VEL
LIN {X 0,Y 283.613,Z 531.468,A -85,B 0,C 180,E1 -16996.385,E2 -16996.385} C_VEL
LIN {X 0,Y 282.782,Z 537.041,A -85,B 0,C 180,E1 -16999.258,E2 -16999.258} C_VEL
LIN {X 0,Y 282.527,Z 540.263,A -85,B 0,C 180,E1 -17001.417,E2 -17001.417} C_VEL
LIN {X 0,Y 282.434,Z 543.582,A -85,B 0,C 180,E1 -17004.469,E2 -17004.469} C_VEL
LIN {X 0,Y 282.441,Z 545.32,A -85,B 0,C 180,E1 -17007.148,E2 -17007.148} C_VEL
LIN {X 0,Y 282.489,Z 545.956,A -85,B 0,C 180,E1 -17010.001,E2 -17010.001} C_VEL
LIN {X 0,Y 282.451,Z 545.309,A -85,B 0,C 180,E1 -17012.853,E2 -17012.853} C_VEL
LIN {X 0,Y 282.463,Z 543.408,A -85,B 0,C 180,E1 -17015.712,E2 -17015.712} C_VEL
LIN {X 0,Y 282.547,Z 540.228,A -85,B 0,C 180,E1 -17018.583,E2 -17018.583} C_VEL
LIN {X 0,Y 282.944,Z 535.708,A -85,B 0,C 180,E1 -17021.462,E2 -17021.462} C_VEL
LIN {X 0,Y 283.947,Z 529.742,A -85,B 0,C 180,E1 -17024.331,E2 -17024.331} C_VEL
LIN {X 0,Y 285.376,Z 522.164,A -85,B 0,C 180,E1 -17027.189,E2 -17027.189} C_VEL
LIN {X 0,Y 287.058,Z 514.008,A -85,B 0,C 180,E1 -17029.673,E2 -17029.673} C_VEL
LIN {X 0,Y 289.012,Z 505.699,A -85,B 0,C 180,E1 -17031.768,E2 -17031.768} C_VEL
LIN {X 0,Y 291.098,Z 495.851,A -85,B 0,C 180,E1 -17033.863,E2 -17033.863} C_VEL
LIN {X 0,Y 293.697,Z 484.21,A -85,B 0,C 180,E1 -17035.894,E2 -17035.894} C_VEL
LIN {X 0,Y 296.215,Z 472.584,A -85,B 0,C 180,E1 -17037.559,E2 -17037.559} C_VEL
LIN {X 0,Y 298.711,Z 460.021,A -85,B 0,C 180,E1 -17039.03,E2 -17039.03} C_VEL
LIN {X 0,Y 300.852,Z 447.284,A -85,B 0,C 180,E1 -17040.248,E2 -17040.248} C_VEL
LIN {X 0,Y 302.861,Z 433.524,A -85,B 0,C 180,E1 -17041.28,E2 -17041.28} C_VEL
LIN {X 0,Y 304.652,Z 418.879,A -85,B 0,C 180,E1 -17042.094,E2 -17042.094} C_VEL
LIN {X 0,Y 305.919,Z 403.842,A -85,B 0,C 180,E1 -17042.675,E2 -17042.675} C_VEL
LIN {X 0,Y 310.46,Z 289.481,A -85,B 0,C 180,E1 -17045.418,E2 -17045.418} C_VEL
LIN {X 0,Y 308.407,Z 275.493,A -85,B 0,C 180,E1 -17046.075,E2 -17046.075} C_VEL
LIN {X 0,Y 299.5,Z 256.717,A -85,B 0,C 180,E1 -17047.823,E2 -17047.823} C_VEL
LIN {X 0,Y 293.369,Z 244.924,A -85,B 0,C 180,E1 -17049.115,E2 -17049.115} C_VEL
LIN {X 0,Y 290.621,Z 235.65,A -85,B 0,C 180,E1 -17051.96,E2 -17051.96} C_VEL
LIN {X 0,Y 288.18,Z 228.102,A -85,B 0,C 180,E1 -17054.493,E2 -17054.493} C_VEL
LIN {X 0,Y 285.154,Z 219.322,A -85,B 0,C 180,E1 -17057.679,E2 -17057.679} C_VEL
LIN {X 0,Y 284.291,Z 216.787,A -85,B 0,C 180,E1 -17058.72,E2 -17058.72} C_VEL
LIN {X 0,Y 284.318,Z 216.673,A -85,B 0,C 180,E1 -17062.279,E2 -17062.279} C_VEL
LIN {X 0,Y 284.321,Z 216.69,A -85,B 0,C 180,E1 -17065.353,E2 -17065.353} C_VEL
LIN {X 0,Y 284.294,Z 216.676,A -85,B 0,C 180,E1 -17068.726,E2 -17068.726} C_VEL
LIN {X 0,Y 284.325,Z 216.668,A -85,B 0,C 180,E1 -17071.989,E2 -17071.989} C_VEL
LIN {X 0,Y 284.344,Z 216.67,A -85,B 0,C 180,E1 -17075.154,E2 -17075.154} C_VEL
LIN {X 0,Y 284.326,Z 216.685,A -85,B 0,C 180,E1 -17078.237,E2 -17078.237} C_VEL
LIN {X 0,Y 284.402,Z 216.679,A -85,B 0,C 180,E1 -17081.262,E2 -17081.262} C_VEL
LIN {X 0,Y 284.492,Z 216.672,A -85,B 0,C 180,E1 -17084.459,E2 -17084.459} C_VEL
LIN {X 0,Y 284.486,Z 216.672,A -85,B 0,C 180,E1 -17088.602,E2 -17088.602} C_VEL
LIN {X 0,Y 284.638,Z 216.65,A -85,B 0,C 180,E1 -17091.481,E2 -17091.481} C_VEL
LIN {X 0,Y 284.596,Z 216.647,A -85,B 0,C 180,E1 -17094.331,E2 -17094.331} C_VEL
LIN {X 0,Y 284.854,Z 216.614,A -85,B 0,C 180,E1 -17098.586,E2 -17098.586} C_VEL
LIN {X 0,Y 284.853,Z 216.628,A -85,B 0,C 180,E1 -17101.414,E2 -17101.414} C_VEL
LIN {X 0,Y 284.697,Z 216.636,A -85,B 0,C 180,E1 -17107.09,E2 -17107.09} C_VEL
LIN {X 0,Y 284.566,Z 216.663,A -85,B 0,C 180,E1 -17109.956,E2 -17109.956} C_VEL
LIN {X 0,Y 284.478,Z 216.674,A -85,B 0,C 180,E1 -17114.303,E2 -17114.303} C_VEL
LIN {X 0,Y 284.425,Z 216.676,A -85,B 0,C 180,E1 -17117.249,E2 -17117.249} C_VEL
LIN {X 0,Y 284.38,Z 216.676,A -85,B 0,C 180,E1 -17120.242,E2 -17120.242} C_VEL
LIN {X 0,Y 284.369,Z 216.679,A -85,B 0,C 180,E1 -17123.875,E2 -17123.875} C_VEL
LIN {X 0,Y 284.396,Z 216.662,A -85,B 0,C 180,E1 -17127.173,E2 -17127.173} C_VEL
LIN {X 0,Y 284.294,Z 216.693,A -85,B 0,C 180,E1 -17131.275,E2 -17131.275} C_VEL
LIN {X 0,Y 284.362,Z 216.662,A -85,B 0,C 180,E1 -17135.354,E2 -17135.354} C_VEL
LIN {X 0,Y 284.323,Z 216.686,A -85,B 0,C 180,E1 -17138.168,E2 -17138.168} C_VEL
LIN {X 0,Y 284.271,Z 216.703,A -85,B 0,C 180,E1 -17142.125,E2 -17142.125} C_VEL
LIN {X 0,Y 284.293,Z 216.845,A -85,B 0,C 180,E1 -17143.69,E2 -17143.69} C_VEL
LIN {X 0,Y 287.683,Z 227.207,A -85,B 0,C 180,E1 -17147.801,E2 -17147.801} C_VEL
LIN {X 0,Y 290.386,Z 236.159,A -85,B 0,C 180,E1 -17151.005,E2 -17151.005} C_VEL
LIN {X 0,Y 292.774,Z 244.787,A -85,B 0,C 180,E1 -17153.783,E2 -17153.783} C_VEL
LIN {X 0,Y 301.141,Z 261.136,A -85,B 0,C 180,E1 -17155.482,E2 -17155.482} C_VEL
LIN {X 0,Y 306.546,Z 273.05,A -85,B 0,C 180,E1 -17156.535,E2 -17156.535} C_VEL
LIN {X 0,Y 309.841,Z 291.067,A -85,B 0,C 180,E1 -17157.434,E2 -17157.434} C_VEL
LIN {X 0,Y 306.928,Z 381.691,A -85,B 0,C 180,E1 -17159.418,E2 -17159.418} C_VEL
LIN {X 0,Y 306.208,Z 396.898,A -85,B 0,C 180,E1 -17159.863,E2 -17159.863} C_VEL
LIN {X 0,Y 305.02,Z 410.49,A -85,B 0,C 180,E1 -17160.495,E2 -17160.495} C_VEL
LIN {X 0,Y 303.288,Z 424.932,A -85,B 0,C 180,E1 -17161.449,E2 -17161.449} C_VEL
LIN {X 0,Y 301.456,Z 436.502,A -85,B 0,C 180,E1 -17162.436,E2 -17162.436} C_VEL
LIN {X 0,Y 299.502,Z 448.205,A -85,B 0,C 180,E1 -17163.71,E2 -17163.71} C_VEL
LIN {X 0,Y 297.109,Z 459.346,A -85,B 0,C 180,E1 -17165.174,E2 -17165.174} C_VEL
LIN {X 0,Y 294.776,Z 469.639,A -85,B 0,C 180,E1 -17166.834,E2 -17166.834} C_VEL
LIN {X 0,Y 292.265,Z 479.925,A -85,B 0,C 180,E1 -17168.857,E2 -17168.857} C_VEL
LIN {X 0,Y 290.06,Z 488.432,A -85,B 0,C 180,E1 -17170.901,E2 -17170.901} C_VEL
LIN {X 0,Y 288.326,Z 495.582,A -85,B 0,C 180,E1 -17172.992,E2 -17172.992} C_VEL
LIN {X 0,Y 286.606,Z 501.585,A -85,B 0,C 180,E1 -17175.079,E2 -17175.079} C_VEL
LIN {X 0,Y 284.971,Z 507.99,A -85,B 0,C 180,E1 -17177.899,E2 -17177.899} C_VEL
LIN {X 0,Y 283.859,Z 512.836,A -85,B 0,C 180,E1 -17180.739,E2 -17180.739} C_VEL
LIN {X 0,Y 283.309,Z 515.578,A -85,B 0,C 180,E1 -17182.875,E2 -17182.875} C_VEL
LIN {X 0,Y 282.814,Z 518.049,A -85,B 0,C 180,E1 -17185.724,E2 -17185.724} C_VEL
LIN {X 0,Y 282.53,Z 519.283,A -85,B 0,C 180,E1 -17188.574,E2 -17188.574} C_VEL
LIN {X 0,Y 282.522,Z 519.307,A -85,B 0,C 180,E1 -17191.425,E2 -17191.425} C_VEL
LIN {X 0,Y 282.804,Z 518.123,A -85,B 0,C 180,E1 -17194.275,E2 -17194.275} C_VEL
LIN {X 0,Y 283.278,Z 515.705,A -85,B 0,C 180,E1 -17197.125,E2 -17197.125} C_VEL
LIN {X 0,Y 284.031,Z 511.978,A -85,B 0,C 180,E1 -17199.974,E2 -17199.974} C_VEL
LIN {X 0,Y 285.288,Z 506.814,A -85,B 0,C 180,E1 -17202.809,E2 -17202.809} C_VEL
LIN {X 0,Y 287.056,Z 500.025,A -85,B 0,C 180,E1 -17205.623,E2 -17205.623} C_VEL
LIN {X 0,Y 289.107,Z 492.569,A -85,B 0,C 180,E1 -17208.055,E2 -17208.055} C_VEL
LIN {X 0,Y 291.032,Z 484.858,A -85,B 0,C 180,E1 -17210.127,E2 -17210.127} C_VEL
LIN {X 0,Y 293.472,Z 475.597,A -85,B 0,C 180,E1 -17212.158,E2 -17212.158} C_VEL
LIN {X 0,Y 295.862,Z 465.402,A -85,B 0,C 180,E1 -17214.003,E2 -17214.003} C_VEL
LIN {X 0,Y 298.328,Z 454.225,A -85,B 0,C 180,E1 -17215.649,E2 -17215.649} C_VEL
LIN {X 0,Y 300.685,Z 441.901,A -85,B 0,C 180,E1 -17217.119,E2 -17217.119} C_VEL
LIN {X 0,Y 302.591,Z 430.181,A -85,B 0,C 180,E1 -17218.243,E2 -17218.243} C_VEL
LIN {X 0,Y 304.452,Z 416.134,A -85,B 0,C 180,E1 -17219.28,E2 -17219.28} C_VEL
LIN {X 0,Y 305.852,Z 402.126,A -85,B 0,C 180,E1 -17220.032,E2 -17220.032} C_VEL
LIN {X 0,Y 306.795,Z 387.554,A -85,B 0,C 180,E1 -17220.547,E2 -17220.547} C_VEL
LIN {X 0,Y 309.945,Z 291.366,A -85,B 0,C 180,E1 -17222.668,E2 -17222.668} C_VEL
LIN {X 0,Y 306.338,Z 272.284,A -85,B 0,C 180,E1 -17223.637,E2 -17223.637} C_VEL
LIN {X 0,Y 298.33,Z 255.517,A -85,B 0,C 180,E1 -17225.198,E2 -17225.198} C_VEL
LIN {X 0,Y 292.709,Z 244.579,A -85,B 0,C 180,E1 -17226.382,E2 -17226.382} C_VEL
LIN {X 0,Y 290.33,Z 235.866,A -85,B 0,C 180,E1 -17229.229,E2 -17229.229} C_VEL
LIN {X 0,Y 287.826,Z 227.609,A -85,B 0,C 180,E1 -17232.196,E2 -17232.196} C_VEL
LIN {X 0,Y 284.755,Z 218.508,A -85,B 0,C 180,E1 -17235.757,E2 -17235.757} C_VEL
LIN {X 0,Y 283.96,Z 217.311,A -85,B 0,C 180,E1 -17236.479,E2 -17236.479} C_VEL
LIN {X 0,Y 282.275,Z 216.947,A -85,B 0,C 180,E1 -17237.611,E2 -17237.611} C_VEL
LIN {X 0,Y 278.22,Z 217.485,A -85,B 0,C 180,E1 -17240.361,E2 -17240.361} C_VEL
LIN {X 0,Y 277.269,Z 217.566,A -85,B 0,C 180,E1 -17242.014,E2 -17242.014} C_VEL
LIN {X 0,Y 277.299,Z 217.545,A -85,B 0,C 180,E1 -17244.343,E2 -17244.343} C_VEL
LIN {X 0,Y 277.241,Z 217.575,A -85,B 0,C 180,E1 -17247.836,E2 -17247.836} C_VEL
LIN {X 0,Y 277.267,Z 217.535,A -85,B 0,C 180,E1 -17251.21,E2 -17251.21} C_VEL
LIN {X 0,Y 277.31,Z 217.567,A -85,B 0,C 180,E1 -17254.479,E2 -17254.479} C_VEL
LIN {X 0,Y 277.286,Z 217.568,A -85,B 0,C 180,E1 -17257.655,E2 -17257.655} C_VEL
LIN {X 0,Y 277.341,Z 217.554,A -85,B 0,C 180,E1 -17260.766,E2 -17260.766} C_VEL
LIN {X 0,Y 277.423,Z 217.55,A -85,B 0,C 180,E1 -17265.325,E2 -17265.325} C_VEL
LIN {X 0,Y 277.501,Z 217.542,A -85,B 0,C 180,E1 -17269.788,E2 -17269.788} C_VEL
LIN {X 0,Y 277.647,Z 217.514,A -85,B 0,C 180,E1 -17272.729,E2 -17272.729} C_VEL
LIN {X 0,Y 277.816,Z 217.503,A -85,B 0,C 180,E1 -17278.55,E2 -17278.55} C_VEL
LIN {X 0,Y 277.816,Z 217.491,A -85,B 0,C 180,E1 -17281.449,E2 -17281.449} C_VEL
LIN {X 0,Y 277.647,Z 217.525,A -85,B 0,C 180,E1 -17287.271,E2 -17287.271} C_VEL
LIN {X 0,Y 277.501,Z 217.532,A -85,B 0,C 180,E1 -17290.211,E2 -17290.211} C_VEL
LIN {X 0,Y 277.429,Z 217.544,A -85,B 0,C 180,E1 -17294.674,E2 -17294.674} C_VEL
LIN {X 0,Y 277.339,Z 217.562,A -85,B 0,C 180,E1 -17299.234,E2 -17299.234} C_VEL
LIN {X 0,Y 277.313,Z 217.559,A -85,B 0,C 180,E1 -17304.17,E2 -17304.17} C_VEL
LIN {X 0,Y 277.316,Z 217.534,A -85,B 0,C 180,E1 -17307.504,E2 -17307.504} C_VEL
LIN {X 0,Y 277.267,Z 217.564,A -85,B 0,C 180,E1 -17310.482,E2 -17310.482} C_VEL
LIN {X 0,Y 277.248,Z 217.554,A -85,B 0,C 180,E1 -17313.895,E2 -17313.895} C_VEL
LIN {X 0,Y 277.26,Z 217.55,A -85,B 0,C 180,E1 -17317.47,E2 -17317.47} C_VEL
LIN {X 0,Y 277.288,Z 217.806,A -85,B 0,C 180,E1 -17319.994,E2 -17319.994} C_VEL
LIN {X 0,Y 280.222,Z 226.234,A -85,B 0,C 180,E1 -17323.339,E2 -17323.339} C_VEL
LIN {X 0,Y 284.001,Z 237.653,A -85,B 0,C 180,E1 -17327.409,E2 -17327.409} C_VEL
LIN {X 0,Y 286.251,Z 245.018,A -85,B 0,C 180,E1 -17329.746,E2 -17329.746} C_VEL
LIN {X 0,Y 294.056,Z 259.858,A -85,B 0,C 180,E1 -17331.45,E2 -17331.45} C_VEL
LIN {X 0,Y 301.783,Z 275.99,A -85,B 0,C 180,E1 -17333.029,E2 -17333.029} C_VEL
LIN {X 0,Y 303.163,Z 279.497,A -85,B 0,C 180,E1 -17333.318,E2 -17333.318} C_VEL
LIN {X 0,Y 304.641,Z 290.828,A -85,B 0,C 180,E1 -17333.846,E2 -17333.846} C_VEL
LIN {X 0,Y 299.966,Z 403.716,A -85,B 0,C 180,E1 -17336.594,E2 -17336.594} C_VEL
LIN {X 0,Y 298.646,Z 418.715,A -85,B 0,C 180,E1 -17337.182,E2 -17337.182} C_VEL
LIN {X 0,Y 296.665,Z 434.493,A -85,B 0,C 180,E1 -17338.091,E2 -17338.091} C_VEL
LIN {X 0,Y 294.396,Z 448.979,A -85,B 0,C 180,E1 -17339.224,E2 -17339.224} C_VEL
LIN {X 0,Y 291.901,Z 462.814,A -85,B 0,C 180,E1 -17340.624,E2 -17340.624} C_VEL
LIN {X 0,Y 289.118,Z 476.062,A -85,B 0,C 180,E1 -17342.297,E2 -17342.297} C_VEL
LIN {X 0,Y 286.321,Z 488.113,A -85,B 0,C 180,E1 -17344.172,E2 -17344.172} C_VEL
LIN {X 0,Y 283.741,Z 499.274,A -85,B 0,C 180,E1 -17346.306,E2 -17346.306} C_VEL
LIN {X 0,Y 281.384,Z 509.774,A -85,B 0,C 180,E1 -17348.768,E2 -17348.768} C_VEL
LIN {X 0,Y 279.225,Z 518.593,A -85,B 0,C 180,E1 -17351.283,E2 -17351.283} C_VEL
LIN {X 0,Y 277.641,Z 525.895,A -85,B 0,C 180,E1 -17353.833,E2 -17353.833} C_VEL
LIN {X 0,Y 276.396,Z 532.627,A -85,B 0,C 180,E1 -17356.772,E2 -17356.772} C_VEL
LIN {X 0,Y 275.634,Z 537.842,A -85,B 0,C 180,E1 -17359.719,E2 -17359.719} C_VEL
LIN {X 0,Y 275.35,Z 541.674,A -85,B 0,C 180,E1 -17362.669,E2 -17362.669} C_VEL
LIN {X 0,Y 275.338,Z 543.424,A -85,B 0,C 180,E1 -17364.546,E2 -17364.546} C_VEL
LIN {X 0,Y 275.366,Z 544.988,A -85,B 0,C 180,E1 -17367.075,E2 -17367.075} C_VEL
LIN {X 0,Y 275.405,Z 545.624,A -85,B 0,C 180,E1 -17370.001,E2 -17370.001} C_VEL
LIN {X 0,Y 275.378,Z 544.976,A -85,B 0,C 180,E1 -17372.926,E2 -17372.926} C_VEL
LIN {X 0,Y 275.379,Z 543.073,A -85,B 0,C 180,E1 -17375.86,E2 -17375.86} C_VEL
LIN {X 0,Y 275.459,Z 539.89,A -85,B 0,C 180,E1 -17378.806,E2 -17378.806} C_VEL
LIN {X 0,Y 275.931,Z 535.367,A -85,B 0,C 180,E1 -17381.757,E2 -17381.757} C_VEL
LIN {X 0,Y 277.002,Z 529.397,A -85,B 0,C 180,E1 -17384.698,E2 -17384.698} C_VEL
LIN {X 0,Y 278.501,Z 521.813,A -85,B 0,C 180,E1 -17387.627,E2 -17387.627} C_VEL
LIN {X 0,Y 280.31,Z 513.652,A -85,B 0,C 180,E1 -17390.166,E2 -17390.166} C_VEL
LIN {X 0,Y 282.673,Z 503.812,A -85,B 0,C 180,E1 -17392.667,E2 -17392.667} C_VEL
LIN {X 0,Y 284.945,Z 493.701,A -85,B 0,C 180,E1 -17394.79,E2 -17394.79} C_VEL
LIN {X 0,Y 287.508,Z 482.728,A -85,B 0,C 180,E1 -17396.691,E2 -17396.691} C_VEL
LIN {X 0,Y 290.125,Z 470.853,A -85,B 0,C 180,E1 -17398.385,E2 -17398.385} C_VEL
LIN {X 0,Y 292.805,Z 457.97,A -85,B 0,C 180,E1 -17399.871,E2 -17399.871} C_VEL
LIN {X 0,Y 294.89,Z 445.645,A -85,B 0,C 180,E1 -17401.038,E2 -17401.038} C_VEL
LIN {X 0,Y 296.952,Z 431.647,A -85,B 0,C 180,E1 -17402.075,E2 -17402.075} C_VEL
LIN {X 0,Y 298.706,Z 417.231,A -85,B 0,C 180,E1 -17402.862,E2 -17402.862} C_VEL
LIN {X 0,Y 299.97,Z 402.744,A -85,B 0,C 180,E1 -17403.407,E2 -17403.407} C_VEL
LIN {X 0,Y 304.561,Z 290.721,A -85,B 0,C 180,E1 -17406.133,E2 -17406.133} C_VEL
LIN {X 0,Y 302.79,Z 278.304,A -85,B 0,C 180,E1 -17406.729,E2 -17406.729} C_VEL
LIN {X 0,Y 294.096,Z 259.9,A -85,B 0,C 180,E1 -17408.503,E2 -17408.503} C_VEL
LIN {X 0,Y 286.225,Z 244.984,A -85,B 0,C 180,E1 -17410.218,E2 -17410.218} C_VEL
LIN {X 0,Y 283.193,Z 234.954,A -85,B 0,C 180,E1 -17413.457,E2 -17413.457} C_VEL
LIN {X 0,Y 279.274,Z 223.373,A -85,B 0,C 180,E1 -17417.688,E2 -17417.688} C_VEL
LIN {X 0,Y 277.267,Z 217.65,A -85,B 0,C 180,E1 -17420.057,E2 -17420.057} C_VEL
LIN {X 0,Y 277.295,Z 217.568,A -85,B 0,C 180,E1 -17424.343,E2 -17424.343} C_VEL
LIN {X 0,Y 277.243,Z 217.547,A -85,B 0,C 180,E1 -17427.837,E2 -17427.837} C_VEL
LIN {X 0,Y 277.268,Z 217.561,A -85,B 0,C 180,E1 -17431.21,E2 -17431.21} C_VEL
LIN {X 0,Y 277.31,Z 217.535,A -85,B 0,C 180,E1 -17434.479,E2 -17434.479} C_VEL
LIN {X 0,Y 277.284,Z 217.565,A -85,B 0,C 180,E1 -17437.655,E2 -17437.655} C_VEL
LIN {X 0,Y 277.344,Z 217.562,A -85,B 0,C 180,E1 -17440.766,E2 -17440.766} C_VEL
LIN {X 0,Y 277.434,Z 217.544,A -85,B 0,C 180,E1 -17445.326,E2 -17445.326} C_VEL
LIN {X 0,Y 277.46,Z 217.538,A -85,B 0,C 180,E1 -17449.787,E2 -17449.787} C_VEL
LIN {X 0,Y 277.64,Z 217.526,A -85,B 0,C 180,E1 -17452.729,E2 -17452.729} C_VEL
LIN {X 0,Y 277.82,Z 217.49,A -85,B 0,C 180,E1 -17458.551,E2 -17458.551} C_VEL
LIN {X 0,Y 277.819,Z 217.503,A -85,B 0,C 180,E1 -17461.45,E2 -17461.45} C_VEL
LIN {X 0,Y 277.652,Z 217.513,A -85,B 0,C 180,E1 -17467.271,E2 -17467.271} C_VEL
LIN {X 0,Y 277.506,Z 217.542,A -85,B 0,C 180,E1 -17470.212,E2 -17470.212} C_VEL
LIN {X 0,Y 277.428,Z 217.55,A -85,B 0,C 180,E1 -17474.675,E2 -17474.675} C_VEL
LIN {X 0,Y 277.345,Z 217.554,A -85,B 0,C 180,E1 -17479.234,E2 -17479.234} C_VEL
LIN {X 0,Y 277.329,Z 217.556,A -85,B 0,C 180,E1 -17483.921,E2 -17483.921} C_VEL
LIN {X 0,Y 277.324,Z 217.537,A -85,B 0,C 180,E1 -17487.505,E2 -17487.505} C_VEL
LIN {X 0,Y 277.273,Z 217.55,A -85,B 0,C 180,E1 -17490.482,E2 -17490.482} C_VEL
LIN {X 0,Y 277.254,Z 217.549,A -85,B 0,C 180,E1 -17493.895,E2 -17493.895} C_VEL
LIN {X 0,Y 277.282,Z 217.572,A -85,B 0,C 180,E1 -17497.467,E2 -17497.467} C_VEL
LIN {X 0,Y 277.239,Z 217.576,A -85,B 0,C 180,E1 -17501.988,E2 -17501.988} C_VEL
LIN {X 0,Y 277.262,Z 217.749,A -85,B 0,C 180,E1 -17502.412,E2 -17502.412} C_VEL
LIN {X 0,Y 280.211,Z 226.633,A -85,B 0,C 180,E1 -17506.144,E2 -17506.144} C_VEL
LIN {X 0,Y 283.248,Z 236.369,A -85,B 0,C 180,E1 -17509.826,E2 -17509.826} C_VEL
LIN {X 0,Y 285.56,Z 244.635,A -85,B 0,C 180,E1 -17512.638,E2 -17512.638} C_VEL
LIN {X 0,Y 292.712,Z 258.227,A -85,B 0,C 180,E1 -17514.189,E2 -17514.189} C_VEL
LIN {X 0,Y 300.748,Z 275.002,A -85,B 0,C 180,E1 -17515.814,E2 -17515.814} C_VEL
LIN {X 0,Y 303.939,Z 292.37,A -85,B 0,C 180,E1 -17516.715,E2 -17516.715} C_VEL
LIN {X 0,Y 301.02,Z 379.346,A -85,B 0,C 180,E1 -17518.654,E2 -17518.654} C_VEL
LIN {X 0,Y 300.277,Z 395.507,A -85,B 0,C 180,E1 -17519.106,E2 -17519.106} C_VEL
LIN {X 0,Y 299.035,Z 409.635,A -85,B 0,C 180,E1 -17519.746,E2 -17519.746} C_VEL
LIN {X 0,Y 297.419,Z 423.334,A -85,B 0,C 180,E1 -17520.638,E2 -17520.638} C_VEL
LIN {X 0,Y 295.209,Z 437.002,A -85,B 0,C 180,E1 -17521.805,E2 -17521.805} C_VEL
LIN {X 0,Y 292.884,Z 449.988,A -85,B 0,C 180,E1 -17523.261,E2 -17523.261} C_VEL
LIN {X 0,Y 290.44,Z 460.895,A -85,B 0,C 180,E1 -17524.755,E2 -17524.755} C_VEL
LIN {X 0,Y 287.86,Z 471.899,A -85,B 0,C 180,E1 -17526.625,E2 -17526.625} C_VEL
LIN {X 0,Y 285.244,Z 481.834,A -85,B 0,C 180,E1 -17528.689,E2 -17528.689} C_VEL
LIN {X 0,Y 282.967,Z 490.472,A -85,B 0,C 180,E1 -17530.896,E2 -17530.896} C_VEL
LIN {X 0,Y 280.953,Z 498.075,A -85,B 0,C 180,E1 -17533.281,E2 -17533.281} C_VEL
LIN {X 0,Y 279.258,Z 503.686,A -85,B 0,C 180,E1 -17535.423,E2 -17535.423} C_VEL
LIN {X 0,Y 277.693,Z 509.707,A -85,B 0,C 180,E1 -17538.318,E2 -17538.318} C_VEL
LIN {X 0,Y 276.651,Z 514.193,A -85,B 0,C 180,E1 -17541.232,E2 -17541.232} C_VEL
LIN {X 0,Y 275.967,Z 517.306,A -85,B 0,C 180,E1 -17544.153,E2 -17544.153} C_VEL
LIN {X 0,Y 275.574,Z 519.151,A -85,B 0,C 180,E1 -17547.076,E2 -17547.076} C_VEL
LIN {X 0,Y 275.421,Z 519.777,A -85,B 0,C 180,E1 -17549.999,E2 -17549.999} C_VEL
LIN {X 0,Y 275.553,Z 519.199,A -85,B 0,C 180,E1 -17552.923,E2 -17552.923} C_VEL
LIN {X 0,Y 275.951,Z 517.405,A -85,B 0,C 180,E1 -17555.846,E2 -17555.846} C_VEL
LIN {X 0,Y 276.582,Z 514.345,A -85,B 0,C 180,E1 -17558.769,E2 -17558.769} C_VEL
LIN {X 0,Y 277.646,Z 509.922,A -85,B 0,C 180,E1 -17561.683,E2 -17561.683} C_VEL
LIN {X 0,Y 279.183,Z 503.977,A -85,B 0,C 180,E1 -17564.579,E2 -17564.579} C_VEL
LIN {X 0,Y 281.153,Z 497.378,A -85,B 0,C 180,E1 -17567.08,E2 -17567.08} C_VEL
LIN {X 0,Y 283.054,Z 490.053,A -85,B 0,C 180,E1 -17569.349,E2 -17569.349} C_VEL
LIN {X 0,Y 285.546,Z 480.808,A -85,B 0,C 180,E1 -17571.665,E2 -17571.665} C_VEL
LIN {X 0,Y 288.207,Z 470.635,A -85,B 0,C 180,E1 -17573.725,E2 -17573.725} C_VEL
LIN {X 0,Y 290.892,Z 459.324,A -85,B 0,C 180,E1 -17575.585,E2 -17575.585} C_VEL
LIN {X 0,Y 293.33,Z 448.127,A -85,B 0,C 180,E1 -17577.079,E2 -17577.079} C_VEL
LIN {X 0,Y 295.511,Z 435.973,A -85,B 0,C 180,E1 -17578.401,E2 -17578.401} C_VEL
LIN {X 0,Y 297.549,Z 422.518,A -85,B 0,C 180,E1 -17579.541,E2 -17579.541} C_VEL
LIN {X 0,Y 299.204,Z 408.501,A -85,B 0,C 180,E1 -17580.429,E2 -17580.429} C_VEL
LIN {X 0,Y 300.442,Z 393.797,A -85,B 0,C 180,E1 -17581.069,E2 -17581.069} C_VEL
LIN {X 0,Y 301.293,Z 374.711,A -85,B 0,C 180,E1 -17581.558,E2 -17581.558} C_VEL
LIN {X 0,Y 304.038,Z 292.141,A -85,B 0,C 180,E1 -17583.403,E2 -17583.403} C_VEL
LIN {X 0,Y 300.83,Z 275.167,A -85,B 0,C 180,E1 -17584.296,E2 -17584.296} C_VEL
LIN {X 0,Y 291.943,Z 256.625,A -85,B 0,C 180,E1 -17586.103,E2 -17586.103} C_VEL
LIN {X 0,Y 285.516,Z 244.475,A -85,B 0,C 180,E1 -17587.526,E2 -17587.526} C_VEL
LIN {X 0,Y 282.597,Z 234.038,A -85,B 0,C 180,E1 -17591.16,E2 -17591.16} C_VEL
LIN {X 0,Y 279.254,Z 223.673,A -85,B 0,C 180,E1 -17595.196,E2 -17595.196} C_VEL
LIN {X 0,Y 277.231,Z 217.651,A -85,B 0,C 180,E1 -17597.853,E2 -17597.853} C_VEL
LIN {X 0,Y 277.269,Z 217.566,A -85,B 0,C 180,E1 -17602.014,E2 -17602.014} C_VEL
LIN {X 0,Y 276.591,Z 217.661,A -85,B 0,C 180,E1 -17603.227,E2 -17603.227} C_VEL
LIN {X 0,Y 273.689,Z 218.014,A -85,B 0,C 180,E1 -17605.202,E2 -17605.202} C_VEL
LIN {X 0,Y 271.25,Z 218.307,A -85,B 0,C 180,E1 -17606.807,E2 -17606.807} C_VEL
LIN {X 0,Y 270.236,Z 218.45,A -85,B 0,C 180,E1 -17608.052,E2 -17608.052} C_VEL
LIN {X 0,Y 270.171,Z 218.45,A -85,B 0,C 180,E1 -17608.474,E2 -17608.474} C_VEL
LIN {X 0,Y 270.26,Z 218.411,A -85,B 0,C 180,E1 -17612.145,E2 -17612.145} C_VEL
LIN {X 0,Y 270.273,Z 218.438,A -85,B 0,C 180,E1 -17615.518,E2 -17615.518} C_VEL
LIN {X 0,Y 270.298,Z 218.429,A -85,B 0,C 180,E1 -17620.244,E2 -17620.244} C_VEL
LIN {X 0,Y 270.391,Z 218.421,A -85,B 0,C 180,E1 -17624.934,E2 -17624.934} C_VEL
LIN {X 0,Y 270.436,Z 218.42,A -85,B 0,C 180,E1 -17629.518,E2 -17629.518} C_VEL
LIN {X 0,Y 270.605,Z 218.39,A -85,B 0,C 180,E1 -17632.538,E2 -17632.538} C_VEL
LIN {X 0,Y 270.782,Z 218.379,A -85,B 0,C 180,E1 -17638.512,E2 -17638.512} C_VEL
LIN {X 0,Y 270.782,Z 218.367,A -85,B 0,C 180,E1 -17641.487,E2 -17641.487} C_VEL
LIN {X 0,Y 270.605,Z 218.402,A -85,B 0,C 180,E1 -17647.461,E2 -17647.461} C_VEL
LIN {X 0,Y 270.436,Z 218.414,A -85,B 0,C 180,E1 -17650.481,E2 -17650.481} C_VEL
LIN {X 0,Y 270.397,Z 218.424,A -85,B 0,C 180,E1 -17655.065,E2 -17655.065} C_VEL
LIN {X 0,Y 270.296,Z 218.442,A -85,B 0,C 180,E1 -17659.756,E2 -17659.756} C_VEL
LIN {X 0,Y 270.268,Z 218.425,A -85,B 0,C 180,E1 -17664.586,E2 -17664.586} C_VEL
LIN {X 0,Y 270.264,Z 218.416,A -85,B 0,C 180,E1 -17667.909,E2 -17667.909} C_VEL
LIN {X 0,Y 270.179,Z 218.431,A -85,B 0,C 180,E1 -17671.349,E2 -17671.349} C_VEL
LIN {X 0,Y 270.205,Z 218.45,A -85,B 0,C 180,E1 -17674.905,E2 -17674.905} C_VEL
LIN {X 0,Y 270.242,Z 218.584,A -85,B 0,C 180,E1 -17678.501,E2 -17678.501} C_VEL
LIN {X 0,Y 273.501,Z 227.871,A -85,B 0,C 180,E1 -17682.418,E2 -17682.418} C_VEL
LIN {X 0,Y 276.9,Z 238.137,A -85,B 0,C 180,E1 -17686.243,E2 -17686.243} C_VEL
LIN {X 0,Y 279.068,Z 245.031,A -85,B 0,C 180,E1 -17688.552,E2 -17688.552} C_VEL
LIN {X 0,Y 287.579,Z 260.769,A -85,B 0,C 180,E1 -17690.495,E2 -17690.495} C_VEL
LIN {X 0,Y 295.414,Z 277.041,A -85,B 0,C 180,E1 -17692.174,E2 -17692.174} C_VEL
LIN {X 0,Y 297.593,Z 282.239,A -85,B 0,C 180,E1 -17692.639,E2 -17692.639} C_VEL
LIN {X 0,Y 298.76,Z 292.549,A -85,B 0,C 180,E1 -17693.112,E2 -17693.112} C_VEL
LIN {X 0,Y 293.965,Z 403.999,A -85,B 0,C 180,E1 -17695.871,E2 -17695.871} C_VEL
LIN {X 0,Y 292.605,Z 418.837,A -85,B 0,C 180,E1 -17696.467,E2 -17696.467} C_VEL
LIN {X 0,Y 290.656,Z 433.955,A -85,B 0,C 180,E1 -17697.351,E2 -17697.351} C_VEL
LIN {X 0,Y 288.207,Z 448.956,A -85,B 0,C 180,E1 -17698.54,E2 -17698.54} C_VEL
LIN {X 0,Y 285.682,Z 462.384,A -85,B 0,C 180,E1 -17699.919,E2 -17699.919} C_VEL
LIN {X 0,Y 282.79,Z 475.661,A -85,B 0,C 180,E1 -17701.622,E2 -17701.622} C_VEL
LIN {X 0,Y 279.884,Z 487.732,A -85,B 0,C 180,E1 -17703.532,E2 -17703.532} C_VEL
LIN {X 0,Y 277.211,Z 498.739,A -85,B 0,C 180,E1 -17705.672,E2 -17705.672} C_VEL
LIN {X 0,Y 274.686,Z 509.417,A -85,B 0,C 180,E1 -17708.224,E2 -17708.224} C_VEL
LIN {X 0,Y 272.412,Z 518.243,A -85,B 0,C 180,E1 -17710.796,E2 -17710.796} C_VEL
LIN {X 0,Y 270.749,Z 525.55,A -85,B 0,C 180,E1 -17713.41,E2 -17713.41} C_VEL
LIN {X 0,Y 269.391,Z 532.285,A -85,B 0,C 180,E1 -17716.421,E2 -17716.421} C_VEL
LIN {X 0,Y 268.578,Z 537.503,A -85,B 0,C 180,E1 -17719.446,E2 -17719.446} C_VEL
LIN {X 0,Y 268.269,Z 541.339,A -85,B 0,C 180,E1 -17722.474,E2 -17722.474} C_VEL
LIN {X 0,Y 268.237,Z 543.273,A -85,B 0,C 180,E1 -17724.637,E2 -17724.637} C_VEL
LIN {X 0,Y 268.269,Z 544.654,A -85,B 0,C 180,E1 -17726.997,E2 -17726.997} C_VEL
LIN {X 0,Y 268.323,Z 545.292,A -85,B 0,C 180,E1 -17730.001,E2 -17730.001} C_VEL
LIN {X 0,Y 268.282,Z 544.643,A -85,B 0,C 180,E1 -17733.004,E2 -17733.004} C_VEL
LIN {X 0,Y 268.291,Z 542.738,A -85,B 0,C 180,E1 -17736.015,E2 -17736.015} C_VEL
LIN {X 0,Y 268.392,Z 539.552,A -85,B 0,C 180,E1 -17739.04,E2 -17739.04} C_VEL
LIN {X 0,Y 268.934,Z 535.027,A -85,B 0,C 180,E1 -17742.068,E2 -17742.068} C_VEL
LIN {X 0,Y 270.035,Z 529.051,A -85,B 0,C 180,E1 -17745.086,E2 -17745.086} C_VEL
LIN {X 0,Y 271.645,Z 521.462,A -85,B 0,C 180,E1 -17748.087,E2 -17748.087} C_VEL
LIN {X 0,Y 273.576,Z 513.295,A -85,B 0,C 180,E1 -17750.685,E2 -17750.685} C_VEL
LIN {X 0,Y 275.999,Z 503.72,A -85,B 0,C 180,E1 -17753.176,E2 -17753.176} C_VEL
LIN {X 0,Y 278.451,Z 493.323,A -85,B 0,C 180,E1 -17755.409,E2 -17755.409} C_VEL
LIN {X 0,Y 281.153,Z 482.334,A -85,B 0,C 180,E1 -17757.344,E2 -17757.344} C_VEL
LIN {X 0,Y 283.877,Z 470.433,A -85,B 0,C 180,E1 -17759.069,E2 -17759.069} C_VEL
LIN {X 0,Y 286.642,Z 457.512,A -85,B 0,C 180,E1 -17760.581,E2 -17760.581} C_VEL
LIN {X 0,Y 288.856,Z 444.629,A -85,B 0,C 180,E1 -17761.813,E2 -17761.813} C_VEL
LIN {X 0,Y 291.115,Z 429.751,A -85,B 0,C 180,E1 -17762.901,E2 -17762.901} C_VEL
LIN {X 0,Y 292.949,Z 414.664,A -85,B 0,C 180,E1 -17763.696,E2 -17763.696} C_VEL
LIN {X 0,Y 294.075,Z 400.152,A -85,B 0,C 180,E1 -17764.22,E2 -17764.22} C_VEL
LIN {X 0,Y 298.726,Z 291.786,A -85,B 0,C 180,E1 -17766.88,E2 -17766.88} C_VEL
LIN {X 0,Y 297.223,Z 281.112,A -85,B 0,C 180,E1 -17767.407,E2 -17767.407} C_VEL
LIN {X 0,Y 289.039,Z 263.712,A -85,B 0,C 180,E1 -17769.143,E2 -17769.143} C_VEL
LIN {X 0,Y 280.94,Z 248.503,A -85,B 0,C 180,E1 -17770.935,E2 -17770.935} C_VEL
LIN {X 0,Y 278.996,Z 244.811,A -85,B 0,C 180,E1 -17771.448,E2 -17771.448} C_VEL
LIN {X 0,Y 276.155,Z 235.745,A -85,B 0,C 180,E1 -17774.555,E2 -17774.555} C_VEL
LIN {X 0,Y 272.772,Z 225.814,A -85,B 0,C 180,E1 -17778.347,E2 -17778.347} C_VEL
LIN {X 0,Y 270.211,Z 218.538,A -85,B 0,C 180,E1 -17781.494,E2 -17781.494} C_VEL
LIN {X 0,Y 270.21,Z 218.452,A -85,B 0,C 180,E1 -17785.096,E2 -17785.096} C_VEL
LIN {X 0,Y 270.2,Z 218.436,A -85,B 0,C 180,E1 -17789.131,E2 -17789.131} C_VEL
LIN {X 0,Y 270.262,Z 218.415,A -85,B 0,C 180,E1 -17792.147,E2 -17792.147} C_VEL
LIN {X 0,Y 270.276,Z 218.427,A -85,B 0,C 180,E1 -17795.52,E2 -17795.52} C_VEL
LIN {X 0,Y 270.301,Z 218.442,A -85,B 0,C 180,E1 -17800.245,E2 -17800.245} C_VEL
LIN {X 0,Y 270.402,Z 218.424,A -85,B 0,C 180,E1 -17804.936,E2 -17804.936} C_VEL
LIN {X 0,Y 270.412,Z 218.417,A -85,B 0,C 180,E1 -17809.518,E2 -17809.518} C_VEL
LIN {X 0,Y 270.598,Z 218.403,A -85,B 0,C 180,E1 -17812.539,E2 -17812.539} C_VEL
LIN {X 0,Y 270.786,Z 218.367,A -85,B 0,C 180,E1 -17818.513,E2 -17818.513} C_VEL
LIN {X 0,Y 270.785,Z 218.379,A -85,B 0,C 180,E1 -17821.487,E2 -17821.487} C_VEL
LIN {X 0,Y 270.61,Z 218.389,A -85,B 0,C 180,E1 -17827.461,E2 -17827.461} C_VEL
LIN {X 0,Y 270.441,Z 218.42,A -85,B 0,C 180,E1 -17830.481,E2 -17830.481} C_VEL
LIN {X 0,Y 270.396,Z 218.421,A -85,B 0,C 180,E1 -17835.065,E2 -17835.065} C_VEL
LIN {X 0,Y 270.302,Z 218.429,A -85,B 0,C 180,E1 -17839.756,E2 -17839.756} C_VEL
LIN {X 0,Y 270.274,Z 218.438,A -85,B 0,C 180,E1 -17844.586,E2 -17844.586} C_VEL
LIN {X 0,Y 270.27,Z 218.41,A -85,B 0,C 180,E1 -17847.909,E2 -17847.909} C_VEL
LIN {X 0,Y 270.185,Z 218.45,A -85,B 0,C 180,E1 -17851.348,E2 -17851.348} C_VEL
LIN {X 0,Y 270.215,Z 218.421,A -85,B 0,C 180,E1 -17854.904,E2 -17854.904} C_VEL
LIN {X 0,Y 270.223,Z 218.432,A -85,B 0,C 180,E1 -17858.717,E2 -17858.717} C_VEL
LIN {X 0,Y 270.2,Z 218.688,A -85,B 0,C 180,E1 -17861.036,E2 -17861.036} C_VEL
LIN {X 0,Y 273.264,Z 227.666,A -85,B 0,C 180,E1 -17865.013,E2 -17865.013} C_VEL
LIN {X 0,Y 276.071,Z 236.562,A -85,B 0,C 180,E1 -17868.556,E2 -17868.556} C_VEL
LIN {X 0,Y 278.393,Z 244.666,A -85,B 0,C 180,E1 -17871.443,E2 -17871.443} C_VEL
LIN {X 0,Y 286.182,Z 259.09,A -85,B 0,C 180,E1 -17873.214,E2 -17873.214} C_VEL
LIN {X 0,Y 292.799,Z 272.595,A -85,B 0,C 180,E1 -17874.62,E2 -17874.62} C_VEL
LIN {X 0,Y 295.643,Z 279.201,A -85,B 0,C 180,E1 -17875.22,E2 -17875.22} C_VEL
LIN {X 0,Y 298.12,Z 293.643,A -85,B 0,C 180,E1 -17875.972,E2 -17875.972} C_VEL
LIN {X 0,Y 294.629,Z 390.566,A -85,B 0,C 180,E1 -17878.196,E2 -17878.196} C_VEL
LIN {X 0,Y 293.492,Z 404.932,A -85,B 0,C 180,E1 -17878.763,E2 -17878.763} C_VEL
LIN {X 0,Y 291.894,Z 419.371,A -85,B 0,C 180,E1 -17879.627,E2 -17879.627} C_VEL
LIN {X 0,Y 289.992,Z 431.809,A -85,B 0,C 180,E1 -17880.609,E2 -17880.609} C_VEL
LIN {X 0,Y 287.869,Z 443.936,A -85,B 0,C 180,E1 -17881.842,E2 -17881.842} C_VEL
LIN {X 0,Y 285.275,Z 456.665,A -85,B 0,C 180,E1 -17883.479,E2 -17883.479} C_VEL
LIN {X 0,Y 282.793,Z 466.55,A -85,B 0,C 180,E1 -17885.008,E2 -17885.008} C_VEL
LIN {X 0,Y 280.042,Z 477.457,A -85,B 0,C 180,E1 -17887.108,E2 -17887.108} C_VEL
LIN {X 0,Y 277.411,Z 486.518,A -85,B 0,C 180,E1 -17889.226,E2 -17889.226} C_VEL
LIN {X 0,Y 275.13,Z 495.188,A -85,B 0,C 180,E1 -17891.765,E2 -17891.765} C_VEL
LIN {X 0,Y 272.919,Z 502.268,A -85,B 0,C 180,E1 -17894.312,E2 -17894.312} C_VEL
LIN {X 0,Y 271.079,Z 508.667,A -85,B 0,C 180,E1 -17897.269,E2 -17897.269} C_VEL
LIN {X 0,Y 269.847,Z 513.509,A -85,B 0,C 180,E1 -17900.253,E2 -17900.253} C_VEL
LIN {X 0,Y 269.104,Z 516.667,A -85,B 0,C 180,E1 -17902.943,E2 -17902.943} C_VEL
LIN {X 0,Y 268.705,Z 518.714,A -85,B 0,C 180,E1 -17905.499,E2 -17905.499} C_VEL
LIN {X 0,Y 268.372,Z 519.948,A -85,B 0,C 180,E1 -17908.499,E2 -17908.499} C_VEL
LIN {X 0,Y 268.364,Z 519.971,A -85,B 0,C 180,E1 -17911.5,E2 -17911.5} C_VEL
LIN {X 0,Y 268.695,Z 518.786,A -85,B 0,C 180,E1 -17914.5,E2 -17914.5} C_VEL
LIN {X 0,Y 269.212,Z 516.37,A -85,B 0,C 180,E1 -17917.5,E2 -17917.5} C_VEL
LIN {X 0,Y 270.063,Z 512.646,A -85,B 0,C 180,E1 -17920.495,E2 -17920.495} C_VEL
LIN {X 0,Y 271.448,Z 507.49,A -85,B 0,C 180,E1 -17923.474,E2 -17923.474} C_VEL
LIN {X 0,Y 272.867,Z 502.557,A -85,B 0,C 180,E1 -17925.69,E2 -17925.69} C_VEL
LIN {X 0,Y 275.014,Z 495.544,A -85,B 0,C 180,E1 -17928.242,E2 -17928.242} C_VEL
LIN {X 0,Y 276.952,Z 488.267,A -85,B 0,C 180,E1 -17930.42,E2 -17930.42} C_VEL
LIN {X 0,Y 279.425,Z 479.57,A -85,B 0,C 180,E1 -17932.554,E2 -17932.554} C_VEL
LIN {X 0,Y 282.225,Z 469.087,A -85,B 0,C 180,E1 -17934.651,E2 -17934.651} C_VEL
LIN {X 0,Y 284.814,Z 458.557,A -85,B 0,C 180,E1 -17936.369,E2 -17936.369} C_VEL
LIN {X 0,Y 287.392,Z 446.818,A -85,B 0,C 180,E1 -17937.928,E2 -17937.928} C_VEL
LIN {X 0,Y 289.581,Z 434.684,A -85,B 0,C 180,E1 -17939.236,E2 -17939.236} C_VEL
LIN {X 0,Y 291.705,Z 420.795,A -85,B 0,C 180,E1 -17940.393,E2 -17940.393} C_VEL
LIN {X 0,Y 293.363,Z 406.853,A -85,B 0,C 180,E1 -17941.251,E2 -17941.251} C_VEL
LIN {X 0,Y 294.559,Z 392.369,A -85,B 0,C 180,E1 -17941.862,E2 -17941.862} C_VEL
LIN {X 0,Y 295.709,Z 364.818,A -85,B 0,C 180,E1 -17942.527,E2 -17942.527} C_VEL
LIN {X 0,Y 298.234,Z 293.343,A -85,B 0,C 180,E1 -17944.148,E2 -17944.148} C_VEL
LIN {X 0,Y 295.407,Z 278.223,A -85,B 0,C 180,E1 -17944.968,E2 -17944.968} C_VEL
LIN {X 0,Y 287.303,Z 261.11,A -85,B 0,C 180,E1 -17946.682,E2 -17946.682} C_VEL
LIN {X 0,Y 280.304,Z 248.171,A -85,B 0,C 180,E1 -17948.22,E2 -17948.22} C_VEL
LIN {X 0,Y 278.334,Z 244.408,A -85,B 0,C 180,E1 -17948.746,E2 -17948.746} C_VEL
LIN {X 0,Y 275.517,Z 234.726,A -85,B 0,C 180,E1 -17952.29,E2 -17952.29} C_VEL
LIN {X 0,Y 272.659,Z 225.875,A -85,B 0,C 180,E1 -17955.897,E2 -17955.897} C_VEL
LIN {X 0,Y 270.19,Z 218.522,A -85,B 0,C 180,E1 -17959.267,E2 -17959.267} C_VEL
LIN {X 0,Y 270.235,Z 218.442,A -85,B 0,C 180,E1 -17963.261,E2 -17963.261} C_VEL
LIN {X 0,Y 270.201,Z 218.435,A -85,B 0,C 180,E1 -17966.892,E2 -17966.892} C_VEL
LIN {X 0,Y 270.171,Z 218.45,A -85,B 0,C 180,E1 -17968.474,E2 -17968.474} C_VEL
LIN {X 0,Y 269.547,Z 218.543,A -85,B 0,C 180,E1 -17969.719,E2 -17969.719} C_VEL
LIN {X 0,Y 266.703,Z 218.905,A -85,B 0,C 180,E1 -17971.748,E2 -17971.748} C_VEL
LIN {X 0,Y 264.286,Z 219.199,A -85,B 0,C 180,E1 -17973.398,E2 -17973.398} C_VEL
LIN {X 0,Y 263.281,Z 219.316,A -85,B 0,C 180,E1 -17974.677,E2 -17974.677} C_VEL
LIN {X 0,Y 263.217,Z 219.32,A -85,B 0,C 180,E1 -17975.11,E2 -17975.11} C_VEL
LIN {X 0,Y 263.264,Z 219.306,A -85,B 0,C 180,E1 -17979.693,E2 -17979.693} C_VEL
LIN {X 0,Y 263.34,Z 219.296,A -85,B 0,C 180,E1 -17984.521,E2 -17984.521} C_VEL
LIN {X 0,Y 263.369,Z 219.297,A -85,B 0,C 180,E1 -17989.234,E2 -17989.234} C_VEL
LIN {X 0,Y 263.567,Z 219.266,A -85,B 0,C 180,E1 -17992.338,E2 -17992.338} C_VEL
LIN {X 0,Y 263.746,Z 219.254,A -85,B 0,C 180,E1 -17998.473,E2 -17998.473} C_VEL
LIN {X 0,Y 263.746,Z 219.243,A -85,B 0,C 180,E1 -18001.527,E2 -18001.527} C_VEL
LIN {X 0,Y 263.567,Z 219.28,A -85,B 0,C 180,E1 -18007.661,E2 -18007.661} C_VEL
LIN {X 0,Y 263.368,Z 219.296,A -85,B 0,C 180,E1 -18010.766,E2 -18010.766} C_VEL
LIN {X 0,Y 263.345,Z 219.305,A -85,B 0,C 180,E1 -18015.478,E2 -18015.478} C_VEL
LIN {X 0,Y 263.258,Z 219.314,A -85,B 0,C 180,E1 -18020.307,E2 -18020.307} C_VEL
LIN {X 0,Y 263.202,Z 219.293,A -85,B 0,C 180,E1 -18025.292,E2 -18025.292} C_VEL
LIN {X 0,Y 263.17,Z 219.314,A -85,B 0,C 180,E1 -18028.73,E2 -18028.73} C_VEL
LIN {X 0,Y 263.128,Z 219.302,A -85,B 0,C 180,E1 -18032.289,E2 -18032.289} C_VEL
LIN {X 0,Y 263.165,Z 219.317,A -85,B 0,C 180,E1 -18035.981,E2 -18035.981} C_VEL
LIN {X 0,Y 263.206,Z 219.591,A -85,B 0,C 180,E1 -18037.02,E2 -18037.02} C_VEL
LIN {X 0,Y 266.587,Z 229.011,A -85,B 0,C 180,E1 -18041.229,E2 -18041.229} C_VEL
LIN {X 0,Y 269.555,Z 237.937,A -85,B 0,C 180,E1 -18044.745,E2 -18044.745} C_VEL
LIN {X 0,Y 271.884,Z 245.073,A -85,B 0,C 180,E1 -18047.273,E2 -18047.273} C_VEL
LIN {X 0,Y 279.789,Z 259.211,A -85,B 0,C 180,E1 -18049.183,E2 -18049.183} C_VEL
LIN {X 0,Y 287.3,Z 274.156,A -85,B 0,C 180,E1 -18050.879,E2 -18050.879} C_VEL
LIN {X 0,Y 292.059,Z 285.064,A -85,B 0,C 180,E1 -18051.936,E2 -18051.936} C_VEL
LIN {X 0,Y 292.978,Z 293.64,A -85,B 0,C 180,E1 -18052.336,E2 -18052.336} C_VEL
LIN {X 0,Y 288.093,Z 403.029,A -85,B 0,C 180,E1 -18055.075,E2 -18055.075} C_VEL
LIN {X 0,Y 286.679,Z 418.151,A -85,B 0,C 180,E1 -18055.679,E2 -18055.679} C_VEL
LIN {X 0,Y 284.659,Z 433.415,A -85,B 0,C 180,E1 -18056.574,E2 -18056.574} C_VEL
LIN {X 0,Y 282.278,Z 447.818,A -85,B 0,C 180,E1 -18057.722,E2 -18057.722} C_VEL
LIN {X 0,Y 279.86,Z 460.512,A -85,B 0,C 180,E1 -18059.017,E2 -18059.017} C_VEL
LIN {X 0,Y 276.759,Z 474.071,A -85,B 0,C 180,E1 -18060.737,E2 -18060.737} C_VEL
LIN {X 0,Y 274.003,Z 485.363,A -85,B 0,C 180,E1 -18062.505,E2 -18062.505} C_VEL
LIN {X 0,Y 271.119,Z 496.712,A -85,B 0,C 180,E1 -18064.678,E2 -18064.678} C_VEL
LIN {X 0,Y 268.72,Z 506.248,A -85,B 0,C 180,E1 -18066.903,E2 -18066.903} C_VEL
LIN {X 0,Y 266.223,Z 515.573,A -85,B 0,C 180,E1 -18069.527,E2 -18069.527} C_VEL
LIN {X 0,Y 264.335,Z 523.281,A -85,B 0,C 180,E1 -18072.197,E2 -18072.197} C_VEL
LIN {X 0,Y 262.73,Z 530.441,A -85,B 0,C 180,E1 -18075.279,E2 -18075.279} C_VEL
LIN {X 0,Y 261.686,Z 536.023,A -85,B 0,C 180,E1 -18078.38,E2 -18078.38} C_VEL
LIN {X 0,Y 261.306,Z 539.252,A -85,B 0,C 180,E1 -18080.714,E2 -18080.714} C_VEL
LIN {X 0,Y 261.193,Z 542.43,A -85,B 0,C 180,E1 -18083.822,E2 -18083.822} C_VEL
LIN {X 0,Y 261.176,Z 544.321,A -85,B 0,C 180,E1 -18086.916,E2 -18086.916} C_VEL
LIN {X 0,Y 261.243,Z 544.959,A -85,B 0,C 180,E1 -18090.001,E2 -18090.001} C_VEL
LIN {X 0,Y 261.19,Z 544.31,A -85,B 0,C 180,E1 -18093.085,E2 -18093.085} C_VEL
LIN {X 0,Y 261.195,Z 542.402,A -85,B 0,C 180,E1 -18096.179,E2 -18096.179} C_VEL
LIN {X 0,Y 261.315,Z 539.213,A -85,B 0,C 180,E1 -18099.287,E2 -18099.287} C_VEL
LIN {X 0,Y 261.942,Z 534.687,A -85,B 0,C 180,E1 -18102.395,E2 -18102.395} C_VEL
LIN {X 0,Y 263.102,Z 528.707,A -85,B 0,C 180,E1 -18105.493,E2 -18105.493} C_VEL
LIN {X 0,Y 264.808,Z 521.112,A -85,B 0,C 180,E1 -18108.571,E2 -18108.571} C_VEL
LIN {X 0,Y 266.889,Z 512.941,A -85,B 0,C 180,E1 -18111.228,E2 -18111.228} C_VEL
LIN {X 0,Y 269.314,Z 503.74,A -85,B 0,C 180,E1 -18113.682,E2 -18113.682} C_VEL
LIN {X 0,Y 271.512,Z 494.758,A -85,B 0,C 180,E1 -18115.694,E2 -18115.694} C_VEL
LIN {X 0,Y 274.539,Z 483.022,A -85,B 0,C 180,E1 -18117.852,E2 -18117.852} C_VEL
LIN {X 0,Y 277.667,Z 470.013,A -85,B 0,C 180,E1 -18119.784,E2 -18119.784} C_VEL
LIN {X 0,Y 280.504,Z 457.054,A -85,B 0,C 180,E1 -18121.325,E2 -18121.325} C_VEL
LIN {X 0,Y 282.701,Z 444.774,A -85,B 0,C 180,E1 -18122.52,E2 -18122.52} C_VEL
LIN {X 0,Y 284.973,Z 430.444,A -85,B 0,C 180,E1 -18123.597,E2 -18123.597} C_VEL
LIN {X 0,Y 286.855,Z 415.708,A -85,B 0,C 180,E1 -18124.405,E2 -18124.405} C_VEL
LIN {X 0,Y 288.133,Z 400.491,A -85,B 0,C 180,E1 -18124.974,E2 -18124.974} C_VEL
LIN {X 0,Y 292.875,Z 292.514,A -85,B 0,C 180,E1 -18127.676,E2 -18127.676} C_VEL
LIN {X 0,Y 291.757,Z 284.078,A -85,B 0,C 180,E1 -18128.098,E2 -18128.098} C_VEL
LIN {X 0,Y 283.952,Z 267.374,A -85,B 0,C 180,E1 -18129.82,E2 -18129.82} C_VEL
LIN {X 0,Y 276.359,Z 253.008,A -85,B 0,C 180,E1 -18131.566,E2 -18131.566} C_VEL
LIN {X 0,Y 271.791,Z 244.834,A -85,B 0,C 180,E1 -18132.727,E2 -18132.727} C_VEL
LIN {X 0,Y 268.756,Z 235.463,A -85,B 0,C 180,E1 -18136.134,E2 -18136.134} C_VEL
LIN {X 0,Y 265.826,Z 226.837,A -85,B 0,C 180,E1 -18139.63,E2 -18139.63} C_VEL
LIN {X 0,Y 263.186,Z 219.407,A -85,B 0,C 180,E1 -18143.056,E2 -18143.056} C_VEL
LIN {X 0,Y 263.183,Z 219.31,A -85,B 0,C 180,E1 -18145.891,E2 -18145.891} C_VEL
LIN {X 0,Y 263.147,Z 219.32,A -85,B 0,C 180,E1 -18149.507,E2 -18149.507} C_VEL
LIN {X 0,Y 263.189,Z 219.288,A -85,B 0,C 180,E1 -18153.003,E2 -18153.003} C_VEL
LIN {X 0,Y 263.184,Z 219.326,A -85,B 0,C 180,E1 -18156.387,E2 -18156.387} C_VEL
LIN {X 0,Y 263.263,Z 219.314,A -85,B 0,C 180,E1 -18159.694,E2 -18159.694} C_VEL
LIN {X 0,Y 263.35,Z 219.305,A -85,B 0,C 180,E1 -18164.522,E2 -18164.522} C_VEL
LIN {X 0,Y 263.354,Z 219.298,A -85,B 0,C 180,E1 -18169.234,E2 -18169.234} C_VEL
LIN {X 0,Y 263.558,Z 219.281,A -85,B 0,C 180,E1 -18172.338,E2 -18172.338} C_VEL
LIN {X 0,Y 263.75,Z 219.243,A -85,B 0,C 180,E1 -18178.473,E2 -18178.473} C_VEL
LIN {X 0,Y 263.75,Z 219.255,A -85,B 0,C 180,E1 -18181.527,E2 -18181.527} C_VEL
LIN {X 0,Y 263.572,Z 219.266,A -85,B 0,C 180,E1 -18187.662,E2 -18187.662} C_VEL
LIN {X 0,Y 263.374,Z 219.297,A -85,B 0,C 180,E1 -18190.766,E2 -18190.766} C_VEL
LIN {X 0,Y 263.345,Z 219.296,A -85,B 0,C 180,E1 -18195.479,E2 -18195.479} C_VEL
LIN {X 0,Y 263.269,Z 219.305,A -85,B 0,C 180,E1 -18200.307,E2 -18200.307} C_VEL
LIN {X 0,Y 263.209,Z 219.325,A -85,B 0,C 180,E1 -18205.292,E2 -18205.292} C_VEL
LIN {X 0,Y 263.166,Z 219.291,A -85,B 0,C 180,E1 -18208.731,E2 -18208.731} C_VEL
LIN {X 0,Y 263.134,Z 219.332,A -85,B 0,C 180,E1 -18212.288,E2 -18212.288} C_VEL
LIN {X 0,Y 263.188,Z 219.302,A -85,B 0,C 180,E1 -18215.978,E2 -18215.978} C_VEL
LIN {X 0,Y 263.165,Z 219.507,A -85,B 0,C 180,E1 -18219.484,E2 -18219.484} C_VEL
LIN {X 0,Y 265.996,Z 227.777,A -85,B 0,C 180,E1 -18223.39,E2 -18223.39} C_VEL
LIN {X 0,Y 268.924,Z 236.789,A -85,B 0,C 180,E1 -18227.197,E2 -18227.197} C_VEL
LIN {X 0,Y 271.228,Z 244.69,A -85,B 0,C 180,E1 -18230.161,E2 -18230.161} C_VEL
LIN {X 0,Y 278.981,Z 258.572,A -85,B 0,C 180,E1 -18232.021,E2 -18232.021} C_VEL
LIN {X 0,Y 286.445,Z 273.5,A -85,B 0,C 180,E1 -18233.69,E2 -18233.69} C_VEL
LIN {X 0,Y 290.16,Z 281.929,A -85,B 0,C 180,E1 -18234.503,E2 -18234.503} C_VEL
LIN {X 0,Y 292.352,Z 295.061,A -85,B 0,C 180,E1 -18235.202,E2 -18235.202} C_VEL
LIN {X 0,Y 288.667,Z 391.533,A -85,B 0,C 180,E1 -18237.459,E2 -18237.459} C_VEL
LIN {X 0,Y 287.389,Z 406.378,A -85,B 0,C 180,E1 -18238.073,E2 -18238.073} C_VEL
LIN {X 0,Y 285.812,Z 419.923,A -85,B 0,C 180,E1 -18238.91,E2 -18238.91} C_VEL
LIN {X 0,Y 283.857,Z 432.287,A -85,B 0,C 180,E1 -18239.909,E2 -18239.909} C_VEL
LIN {X 0,Y 281.624,Z 444.51,A -85,B 0,C 180,E1 -18241.18,E2 -18241.18} C_VEL
LIN {X 0,Y 278.951,Z 457.067,A -85,B 0,C 180,E1 -18242.829,E2 -18242.829} C_VEL
LIN {X 0,Y 276.389,Z 466.934,A -85,B 0,C 180,E1 -18244.388,E2 -18244.388} C_VEL
LIN {X 0,Y 273.517,Z 477.823,A -85,B 0,C 180,E1 -18246.53,E2 -18246.53} C_VEL
LIN {X 0,Y 270.774,Z 486.873,A -85,B 0,C 180,E1 -18248.692,E2 -18248.692} C_VEL
LIN {X 0,Y 268.738,Z 494.423,A -85,B 0,C 180,E1 -18250.919,E2 -18250.919} C_VEL
LIN {X 0,Y 266.715,Z 500.729,A -85,B 0,C 180,E1 -18253.151,E2 -18253.151} C_VEL
LIN {X 0,Y 265.069,Z 506.012,A -85,B 0,C 180,E1 -18255.411,E2 -18255.411} C_VEL
LIN {X 0,Y 263.452,Z 511.608,A -85,B 0,C 180,E1 -18258.458,E2 -18258.458} C_VEL
LIN {X 0,Y 262.625,Z 514.865,A -85,B 0,C 180,E1 -18260.76,E2 -18260.76} C_VEL
LIN {X 0,Y 261.85,Z 517.974,A -85,B 0,C 180,E1 -18263.836,E2 -18263.836} C_VEL
LIN {X 0,Y 261.44,Z 519.815,A -85,B 0,C 180,E1 -18266.918,E2 -18266.918} C_VEL
LIN {X 0,Y 261.261,Z 520.442,A -85,B 0,C 180,E1 -18269.999,E2 -18269.999} C_VEL
LIN {X 0,Y 261.421,Z 519.862,A -85,B 0,C 180,E1 -18273.082,E2 -18273.082} C_VEL
LIN {X 0,Y 261.836,Z 518.07,A -85,B 0,C 180,E1 -18276.163,E2 -18276.163} C_VEL
LIN {X 0,Y 262.556,Z 515.012,A -85,B 0,C 180,E1 -18279.241,E2 -18279.241} C_VEL
LIN {X 0,Y 263.751,Z 510.593,A -85,B 0,C 180,E1 -18282.307,E2 -18282.307} C_VEL
LIN {X 0,Y 265.44,Z 504.657,A -85,B 0,C 180,E1 -18285.352,E2 -18285.352} C_VEL
LIN {X 0,Y 267.602,Z 498.067,A -85,B 0,C 180,E1 -18287.973,E2 -18287.973} C_VEL
LIN {X 0,Y 269.927,Z 489.944,A -85,B 0,C 180,E1 -18290.577,E2 -18290.577} C_VEL
LIN {X 0,Y 272.407,Z 481.529,A -85,B 0,C 180,E1 -18292.767,E2 -18292.767} C_VEL
LIN {X 0,Y 275.303,Z 471.383,A -85,B 0,C 180,E1 -18294.91,E2 -18294.91} C_VEL
LIN {X 0,Y 278.202,Z 460.111,A -85,B 0,C 180,E1 -18296.843,E2 -18296.843} C_VEL
LIN {X 0,Y 280.809,Z 448.973,A -85,B 0,C 180,E1 -18298.393,E2 -18298.393} C_VEL
LIN {X 0,Y 283.148,Z 436.906,A -85,B 0,C 180,E1 -18299.762,E2 -18299.762} C_VEL
LIN {X 0,Y 285.348,Z 423.589,A -85,B 0,C 180,E1 -18300.939,E2 -18300.939} C_VEL
LIN {X 0,Y 287.115,Z 409.811,A -85,B 0,C 180,E1 -18301.856,E2 -18301.856} C_VEL
LIN {X 0,Y 288.447,Z 395.594,A -85,B 0,C 180,E1 -18302.516,E2 -18302.516} C_VEL
LIN {X 0,Y 289.3,Z 379.295,A -85,B 0,C 180,E1 -18302.977,E2 -18302.977} C_VEL
LIN {X 0,Y 292.44,Z 294.63,A -85,B 0,C 180,E1 -18304.926,E2 -18304.926} C_VEL
LIN {X 0,Y 289.885,Z 281.048,A -85,B 0,C 180,E1 -18305.693,E2 -18305.693} C_VEL
LIN {X 0,Y 282.354,Z 265.003,A -85,B 0,C 180,E1 -18307.353,E2 -18307.353} C_VEL
LIN {X 0,Y 275.519,Z 252.3,A -85,B 0,C 180,E1 -18308.915,E2 -18308.915} C_VEL
LIN {X 0,Y 271.189,Z 244.527,A -85,B 0,C 180,E1 -18310.013,E2 -18310.013} C_VEL
LIN {X 0,Y 268.612,Z 235.774,A -85,B 0,C 180,E1 -18313.36,E2 -18313.36} C_VEL
LIN {X 0,Y 265.782,Z 227.059,A -85,B 0,C 180,E1 -18317.086,E2 -18317.086} C_VEL
LIN {X 0,Y 263.162,Z 219.421,A -85,B 0,C 180,E1 -18320.755,E2 -18320.755} C_VEL
LIN {X 0,Y 263.184,Z 219.306,A -85,B 0,C 180,E1 -18324.021,E2 -18324.021} C_VEL
LIN {X 0,Y 263.13,Z 219.33,A -85,B 0,C 180,E1 -18327.711,E2 -18327.711} C_VEL
LIN {X 0,Y 263.192,Z 219.288,A -85,B 0,C 180,E1 -18331.784,E2 -18331.784} C_VEL
LIN {X 0,Y 263.217,Z 219.32,A -85,B 0,C 180,E1 -18335.11,E2 -18335.11} C_VEL
LIN {X 0,Y 262.588,Z 219.396,A -85,B 0,C 180,E1 -18336.388,E2 -18336.388} C_VEL
LIN {X 0,Y 259.716,Z 219.76,A -85,B 0,C 180,E1 -18338.469,E2 -18338.469} C_VEL
LIN {X 0,Y 257.268,Z 220.056,A -85,B 0,C 180,E1 -18340.162,E2 -18340.162} C_VEL
LIN {X 0,Y 256.244,Z 220.188,A -85,B 0,C 180,E1 -18341.476,E2 -18341.476} C_VEL
LIN {X 0,Y 256.176,Z 220.193,A -85,B 0,C 180,E1 -18341.921,E2 -18341.921} C_VEL
LIN {X 0,Y 256.29,Z 220.173,A -85,B 0,C 180,E1 -18344.084,E2 -18344.084} C_VEL
LIN {X 0,Y 256.304,Z 220.174,A -85,B 0,C 180,E1 -18348.933,E2 -18348.933} C_VEL
LIN {X 0,Y 256.535,Z 220.143,A -85,B 0,C 180,E1 -18352.127,E2 -18352.127} C_VEL
LIN {X 0,Y 256.709,Z 220.13,A -85,B 0,C 180,E1 -18358.431,E2 -18358.431} C_VEL
LIN {X 0,Y 256.709,Z 220.119,A -85,B 0,C 180,E1 -18361.569,E2 -18361.569} C_VEL
LIN {X 0,Y 256.534,Z 220.157,A -85,B 0,C 180,E1 -18367.873,E2 -18367.873} C_VEL
LIN {X 0,Y 256.304,Z 220.179,A -85,B 0,C 180,E1 -18371.066,E2 -18371.066} C_VEL
LIN {X 0,Y 256.295,Z 220.186,A -85,B 0,C 180,E1 -18375.915,E2 -18375.915} C_VEL
LIN {X 0,Y 256.161,Z 220.192,A -85,B 0,C 180,E1 -18380.895,E2 -18380.895} C_VEL
LIN {X 0,Y 256.183,Z 220.169,A -85,B 0,C 180,E1 -18385.138,E2 -18385.138} C_VEL
LIN {X 0,Y 256.106,Z 220.21,A -85,B 0,C 180,E1 -18389.6,E2 -18389.6} C_VEL
LIN {X 0,Y 256.08,Z 220.182,A -85,B 0,C 180,E1 -18393.291,E2 -18393.291} C_VEL
LIN {X 0,Y 256.13,Z 220.457,A -85,B 0,C 180,E1 -18395.305,E2 -18395.305} C_VEL
LIN {X 0,Y 258.672,Z 227.362,A -85,B 0,C 180,E1 -18398.675,E2 -18398.675} C_VEL
LIN {X 0,Y 261.517,Z 235.46,A -85,B 0,C 180,E1 -18402.21,E2 -18402.21} C_VEL
LIN {X 0,Y 264.601,Z 244.991,A -85,B 0,C 180,E1 -18405.866,E2 -18405.866} C_VEL
LIN {X 0,Y 272.76,Z 259.101,A -85,B 0,C 180,E1 -18407.957,E2 -18407.957} C_VEL
LIN {X 0,Y 279.432,Z 272.088,A -85,B 0,C 180,E1 -18409.553,E2 -18409.553} C_VEL
LIN {X 0,Y 286.285,Z 286.871,A -85,B 0,C 180,E1 -18411.13,E2 -18411.13} C_VEL
LIN {X 0,Y 287.221,Z 293.128,A -85,B 0,C 180,E1 -18411.473,E2 -18411.473} C_VEL
LIN {X 0,Y 282.205,Z 403.353,A -85,B 0,C 180,E1 -18414.291,E2 -18414.291} C_VEL
LIN {X 0,Y 280.639,Z 419.051,A -85,B 0,C 180,E1 -18414.942,E2 -18414.942} C_VEL
LIN {X 0,Y 278.562,Z 434.008,A -85,B 0,C 180,E1 -18415.851,E2 -18415.851} C_VEL
LIN {X 0,Y 276.063,Z 448.421,A -85,B 0,C 180,E1 -18417.035,E2 -18417.035} C_VEL
LIN {X 0,Y 273.396,Z 461.706,A -85,B 0,C 180,E1 -18418.442,E2 -18418.442} C_VEL
LIN {X 0,Y 270.234,Z 474.859,A -85,B 0,C 180,E1 -18420.174,E2 -18420.174} C_VEL
LIN {X 0,Y 267.114,Z 486.972,A -85,B 0,C 180,E1 -18422.16,E2 -18422.16} C_VEL
LIN {X 0,Y 264.184,Z 498.007,A -85,B 0,C 180,E1 -18424.388,E2 -18424.388} C_VEL
LIN {X 0,Y 261.752,Z 507.318,A -85,B 0,C 180,E1 -18426.67,E2 -18426.67} C_VEL
LIN {X 0,Y 259.496,Z 515.22,A -85,B 0,C 180,E1 -18428.971,E2 -18428.971} C_VEL
LIN {X 0,Y 257.492,Z 522.934,A -85,B 0,C 180,E1 -18431.708,E2 -18431.708} C_VEL
LIN {X 0,Y 255.793,Z 530.098,A -85,B 0,C 180,E1 -18434.871,E2 -18434.871} C_VEL
LIN {X 0,Y 254.69,Z 535.685,A -85,B 0,C 180,E1 -18438.057,E2 -18438.057} C_VEL
LIN {X 0,Y 254.249,Z 538.915,A -85,B 0,C 180,E1 -18440.454,E2 -18440.454} C_VEL
LIN {X 0,Y 254.102,Z 542.096,A -85,B 0,C 180,E1 -18443.649,E2 -18443.649} C_VEL
LIN {X 0,Y 254.086,Z 543.988,A -85,B 0,C 180,E1 -18446.829,E2 -18446.829} C_VEL
LIN {X 0,Y 254.166,Z 544.627,A -85,B 0,C 180,E1 -18450.001,E2 -18450.001} C_VEL
LIN {X 0,Y 254.1,Z 543.976,A -85,B 0,C 180,E1 -18453.172,E2 -18453.172} C_VEL
LIN {X 0,Y 254.104,Z 542.066,A -85,B 0,C 180,E1 -18456.352,E2 -18456.352} C_VEL
LIN {X 0,Y 254.257,Z 538.876,A -85,B 0,C 180,E1 -18459.547,E2 -18459.547} C_VEL
LIN {X 0,Y 254.957,Z 534.347,A -85,B 0,C 180,E1 -18462.74,E2 -18462.74} C_VEL
LIN {X 0,Y 256.174,Z 528.361,A -85,B 0,C 180,E1 -18465.923,E2 -18465.923} C_VEL
LIN {X 0,Y 258.003,Z 520.763,A -85,B 0,C 180,E1 -18469.08,E2 -18469.08} C_VEL
LIN {X 0,Y 260.235,Z 512.587,A -85,B 0,C 180,E1 -18471.798,E2 -18471.798} C_VEL
LIN {X 0,Y 262.555,Z 504.077,A -85,B 0,C 180,E1 -18474.136,E2 -18474.136} C_VEL
LIN {X 0,Y 265.063,Z 494.38,A -85,B 0,C 180,E1 -18476.367,E2 -18476.367} C_VEL
LIN {X 0,Y 268.242,Z 482.628,A -85,B 0,C 180,E1 -18478.565,E2 -18478.565} C_VEL
LIN {X 0,Y 271.175,Z 470.899,A -85,B 0,C 180,E1 -18480.357,E2 -18480.357} C_VEL
LIN {X 0,Y 274.015,Z 458.631,A -85,B 0,C 180,E1 -18481.878,E2 -18481.878} C_VEL
LIN {X 0,Y 276.364,Z 446.256,A -85,B 0,C 180,E1 -18483.144,E2 -18483.144} C_VEL
LIN {X 0,Y 278.713,Z 432.428,A -85,B 0,C 180,E1 -18484.238,E2 -18484.238} C_VEL
LIN {X 0,Y 280.718,Z 417.661,A -85,B 0,C 180,E1 -18485.103,E2 -18485.103} C_VEL
LIN {X 0,Y 282.164,Z 402.298,A -85,B 0,C 180,E1 -18485.716,E2 -18485.716} C_VEL
LIN {X 0,Y 287.16,Z 293.604,A -85,B 0,C 180,E1 -18488.481,E2 -18488.481} C_VEL
LIN {X 0,Y 286.276,Z 286.935,A -85,B 0,C 180,E1 -18488.827,E2 -18488.827} C_VEL
LIN {X 0,Y 278.681,Z 270.537,A -85,B 0,C 180,E1 -18490.576,E2 -18490.576} C_VEL
LIN {X 0,Y 271.389,Z 256.754,A -85,B 0,C 180,E1 -18492.323,E2 -18492.323} C_VEL
LIN {X 0,Y 264.608,Z 244.914,A -85,B 0,C 180,E1 -18494.087,E2 -18494.087} C_VEL
LIN {X 0,Y 261.121,Z 234.244,A -85,B 0,C 180,E1 -18498.231,E2 -18498.231} C_VEL
LIN {X 0,Y 258.64,Z 227.193,A -85,B 0,C 180,E1 -18501.32,E2 -18501.32} C_VEL
LIN {X 0,Y 256.116,Z 220.273,A -85,B 0,C 180,E1 -18504.753,E2 -18504.753} C_VEL
LIN {X 0,Y 256.092,Z 220.184,A -85,B 0,C 180,E1 -18508.573,E2 -18508.573} C_VEL
LIN {X 0,Y 256.138,Z 220.172,A -85,B 0,C 180,E1 -18512.196,E2 -18512.196} C_VEL
LIN {X 0,Y 256.167,Z 220.185,A -85,B 0,C 180,E1 -18515.699,E2 -18515.699} C_VEL
LIN {X 0,Y 256.166,Z 220.192,A -85,B 0,C 180,E1 -18519.105,E2 -18519.105} C_VEL
LIN {X 0,Y 256.3,Z 220.186,A -85,B 0,C 180,E1 -18524.085,E2 -18524.085} C_VEL
LIN {X 0,Y 256.297,Z 220.18,A -85,B 0,C 180,E1 -18528.934,E2 -18528.934} C_VEL
LIN {X 0,Y 256.515,Z 220.159,A -85,B 0,C 180,E1 -18532.127,E2 -18532.127} C_VEL
LIN {X 0,Y 256.497,Z 220.16,A -85,B 0,C 180,E1 -18536.859,E2 -18536.859} C_VEL
LIN {X 0,Y 256.757,Z 220.119,A -85,B 0,C 180,E1 -18540,E2 -18540} C_VEL
LIN {X 0,Y 256.497,Z 220.146,A -85,B 0,C 180,E1 -18543.142,E2 -18543.142} C_VEL
LIN {X 0,Y 256.54,Z 220.142,A -85,B 0,C 180,E1 -18547.873,E2 -18547.873} C_VEL
LIN {X 0,Y 256.31,Z 220.173,A -85,B 0,C 180,E1 -18551.066,E2 -18551.066} C_VEL
LIN {X 0,Y 256.295,Z 220.172,A -85,B 0,C 180,E1 -18555.916,E2 -18555.916} C_VEL
LIN {X 0,Y 256.218,Z 220.187,A -85,B 0,C 180,E1 -18560.891,E2 -18560.891} C_VEL
LIN {X 0,Y 256.189,Z 220.198,A -85,B 0,C 180,E1 -18565.139,E2 -18565.139} C_VEL
LIN {X 0,Y 256.104,Z 220.173,A -85,B 0,C 180,E1 -18569.601,E2 -18569.601} C_VEL
LIN {X 0,Y 256.086,Z 220.19,A -85,B 0,C 180,E1 -18573.29,E2 -18573.29} C_VEL
LIN {X 0,Y 256.137,Z 220.248,A -85,B 0,C 180,E1 -18577.635,E2 -18577.635} C_VEL
LIN {X 0,Y 256.86,Z 222.612,A -85,B 0,C 180,E1 -18578.999,E2 -18578.999} C_VEL
LIN {X 0,Y 259.803,Z 231.009,A -85,B 0,C 180,E1 -18583.081,E2 -18583.081} C_VEL
LIN {X 0,Y 262.699,Z 239.99,A -85,B 0,C 180,E1 -18586.977,E2 -18586.977} C_VEL
LIN {X 0,Y 264.145,Z 244.768,A -85,B 0,C 180,E1 -18588.805,E2 -18588.805} C_VEL
LIN {X 0,Y 272.294,Z 259.121,A -85,B 0,C 180,E1 -18590.871,E2 -18590.871} C_VEL
LIN {X 0,Y 279.703,Z 273.552,A -85,B 0,C 180,E1 -18592.613,E2 -18592.613} C_VEL
LIN {X 0,Y 284.766,Z 284.92,A -85,B 0,C 180,E1 -18593.773,E2 -18593.773} C_VEL
LIN {X 0,Y 286.631,Z 295.906,A -85,B 0,C 180,E1 -18594.384,E2 -18594.384} C_VEL
LIN {X 0,Y 282.805,Z 391.295,A -85,B 0,C 180,E1 -18596.645,E2 -18596.645} C_VEL
LIN {X 0,Y 281.598,Z 405.515,A -85,B 0,C 180,E1 -18597.23,E2 -18597.23} C_VEL
LIN {X 0,Y 279.976,Z 419.341,A -85,B 0,C 180,E1 -18598.081,E2 -18598.081} C_VEL
LIN {X 0,Y 277.758,Z 432.764,A -85,B 0,C 180,E1 -18599.177,E2 -18599.177} C_VEL
LIN {X 0,Y 275.401,Z 445.164,A -85,B 0,C 180,E1 -18600.499,E2 -18600.499} C_VEL
LIN {X 0,Y 272.682,Z 457.466,A -85,B 0,C 180,E1 -18602.151,E2 -18602.151} C_VEL
LIN {X 0,Y 270.028,Z 467.315,A -85,B 0,C 180,E1 -18603.739,E2 -18603.739} C_VEL
LIN {X 0,Y 267.011,Z 478.188,A -85,B 0,C 180,E1 -18605.922,E2 -18605.922} C_VEL
LIN {X 0,Y 264.188,Z 487.226,A -85,B 0,C 180,E1 -18608.134,E2 -18608.134} C_VEL
LIN {X 0,Y 262.024,Z 494.774,A -85,B 0,C 180,E1 -18610.41,E2 -18610.41} C_VEL
LIN {X 0,Y 259.932,Z 501.073,A -85,B 0,C 180,E1 -18612.697,E2 -18612.697} C_VEL
LIN {X 0,Y 258.177,Z 506.353,A -85,B 0,C 180,E1 -18615.012,E2 -18615.012} C_VEL
LIN {X 0,Y 256.495,Z 511.945,A -85,B 0,C 180,E1 -18618.141,E2 -18618.141} C_VEL
LIN {X 0,Y 255.613,Z 515.2,A -85,B 0,C 180,E1 -18620.504,E2 -18620.504} C_VEL
LIN {X 0,Y 254.802,Z 518.308,A -85,B 0,C 180,E1 -18623.665,E2 -18623.665} C_VEL
LIN {X 0,Y 254.377,Z 520.148,A -85,B 0,C 180,E1 -18626.832,E2 -18626.832} C_VEL
LIN {X 0,Y 254.183,Z 520.774,A -85,B 0,C 180,E1 -18629.999,E2 -18629.999} C_VEL
LIN {X 0,Y 254.358,Z 520.194,A -85,B 0,C 180,E1 -18633.167,E2 -18633.167} C_VEL
LIN {X 0,Y 254.772,Z 518.403,A -85,B 0,C 180,E1 -18636.334,E2 -18636.334} C_VEL
LIN {X 0,Y 255.561,Z 515.344,A -85,B 0,C 180,E1 -18639.497,E2 -18639.497} C_VEL
LIN {X 0,Y 256.804,Z 510.929,A -85,B 0,C 180,E1 -18642.646,E2 -18642.646} C_VEL
LIN {X 0,Y 258.589,Z 504.997,A -85,B 0,C 180,E1 -18645.77,E2 -18645.77} C_VEL
LIN {X 0,Y 260.864,Z 498.41,A -85,B 0,C 180,E1 -18648.454,E2 -18648.454} C_VEL
LIN {X 0,Y 263.283,Z 490.294,A -85,B 0,C 180,E1 -18651.121,E2 -18651.121} C_VEL
LIN {X 0,Y 265.894,Z 481.888,A -85,B 0,C 180,E1 -18653.357,E2 -18653.357} C_VEL
LIN {X 0,Y 268.886,Z 471.757,A -85,B 0,C 180,E1 -18655.547,E2 -18655.547} C_VEL
LIN {X 0,Y 271.899,Z 460.504,A -85,B 0,C 180,E1 -18657.517,E2 -18657.517} C_VEL
LIN {X 0,Y 274.609,Z 449.394,A -85,B 0,C 180,E1 -18659.094,E2 -18659.094} C_VEL
LIN {X 0,Y 277.026,Z 437.372,A -85,B 0,C 180,E1 -18660.489,E2 -18660.489} C_VEL
LIN {X 0,Y 279.317,Z 424.122,A -85,B 0,C 180,E1 -18661.683,E2 -18661.683} C_VEL
LIN {X 0,Y 281.152,Z 410.462,A -85,B 0,C 180,E1 -18662.614,E2 -18662.614} C_VEL
LIN {X 0,Y 282.527,Z 396.487,A -85,B 0,C 180,E1 -18663.285,E2 -18663.285} C_VEL
LIN {X 0,Y 283.416,Z 380.635,A -85,B 0,C 180,E1 -18663.752,E2 -18663.752} C_VEL
LIN {X 0,Y 286.708,Z 295.812,A -85,B 0,C 180,E1 -18665.738,E2 -18665.738} C_VEL
LIN {X 0,Y 284.576,Z 284.152,A -85,B 0,C 180,E1 -18666.413,E2 -18666.413} C_VEL
LIN {X 0,Y 277.17,Z 268.39,A -85,B 0,C 180,E1 -18668.111,E2 -18668.111} C_VEL
LIN {X 0,Y 271.443,Z 257.514,A -85,B 0,C 180,E1 -18669.476,E2 -18669.476} C_VEL
LIN {X 0,Y 265.494,Z 247.389,A -85,B 0,C 180,E1 -18670.951,E2 -18670.951} C_VEL
LIN {X 0,Y 263.973,Z 244.379,A -85,B 0,C 180,E1 -18671.441,E2 -18671.441} C_VEL
LIN {X 0,Y 261.443,Z 236.002,A -85,B 0,C 180,E1 -18674.862,E2 -18674.862} C_VEL
LIN {X 0,Y 258.87,Z 228.409,A -85,B 0,C 180,E1 -18678.306,E2 -18678.306} C_VEL
LIN {X 0,Y 256.155,Z 220.306,A -85,B 0,C 180,E1 -18682.429,E2 -18682.429} C_VEL
LIN {X 0,Y 256.082,Z 220.189,A -85,B 0,C 180,E1 -18686.709,E2 -18686.709} C_VEL
LIN {X 0,Y 256.123,Z 220.167,A -85,B 0,C 180,E1 -18691.409,E2 -18691.409} C_VEL
LIN {X 0,Y 256.164,Z 220.193,A -85,B 0,C 180,E1 -18695.698,E2 -18695.698} C_VEL
LIN {X 0,Y 256.214,Z 220.188,A -85,B 0,C 180,E1 -18699.109,E2 -18699.109} C_VEL
LIN {X 0,Y 256.176,Z 220.193,A -85,B 0,C 180,E1 -18701.921,E2 -18701.921} C_VEL
LIN {X 0,Y 255.549,Z 220.278,A -85,B 0,C 180,E1 -18703.233,E2 -18703.233} C_VEL
LIN {X 0,Y 252.722,Z 220.627,A -85,B 0,C 180,E1 -18705.373,E2 -18705.373} C_VEL
LIN {X 0,Y 250.32,Z 220.922,A -85,B 0,C 180,E1 -18707.115,E2 -18707.115} C_VEL
LIN {X 0,Y 249.321,Z 221.041,A -85,B 0,C 180,E1 -18708.466,E2 -18708.466} C_VEL
LIN {X 0,Y 249.257,Z 221.05,A -85,B 0,C 180,E1 -18708.923,E2 -18708.923} C_VEL
LIN {X 0,Y 249.476,Z 221.022,A -85,B 0,C 180,E1 -18711.902,E2 -18711.902} C_VEL
LIN {X 0,Y 249.431,Z 221.026,A -85,B 0,C 180,E1 -18716.769,E2 -18716.769} C_VEL
LIN {X 0,Y 249.723,Z 220.995,A -85,B 0,C 180,E1 -18720,E2 -18720} C_VEL
LIN {X 0,Y 249.432,Z 221.04,A -85,B 0,C 180,E1 -18723.23,E2 -18723.23} C_VEL
LIN {X 0,Y 249.476,Z 221.033,A -85,B 0,C 180,E1 -18728.097,E2 -18728.097} C_VEL
LIN {X 0,Y 249.247,Z 221.062,A -85,B 0,C 180,E1 -18731.383,E2 -18731.383} C_VEL
LIN {X 0,Y 249.237,Z 221.061,A -85,B 0,C 180,E1 -18736.378,E2 -18736.378} C_VEL
LIN {X 0,Y 249.082,Z 221.073,A -85,B 0,C 180,E1 -18741.518,E2 -18741.518} C_VEL
LIN {X 0,Y 249.125,Z 221.043,A -85,B 0,C 180,E1 -18745.482,E2 -18745.482} C_VEL
LIN {X 0,Y 249.075,Z 221.072,A -85,B 0,C 180,E1 -18748.992,E2 -18748.992} C_VEL
LIN {X 0,Y 249.069,Z 221.262,A -85,B 0,C 180,E1 -18753.383,E2 -18753.383} C_VEL
LIN {X 0,Y 251.596,Z 227.866,A -85,B 0,C 180,E1 -18756.911,E2 -18756.911} C_VEL
LIN {X 0,Y 255.017,Z 237.636,A -85,B 0,C 180,E1 -18761.408,E2 -18761.408} C_VEL
LIN {X 0,Y 257.448,Z 245.125,A -85,B 0,C 180,E1 -18764.393,E2 -18764.393} C_VEL
LIN {X 0,Y 265.859,Z 259.252,A -85,B 0,C 180,E1 -18766.674,E2 -18766.674} C_VEL
LIN {X 0,Y 273.414,Z 273.602,A -85,B 0,C 180,E1 -18768.576,E2 -18768.576} C_VEL
LIN {X 0,Y 280.578,Z 289.073,A -85,B 0,C 180,E1 -18770.304,E2 -18770.304} C_VEL
LIN {X 0,Y 281.153,Z 290.485,A -85,B 0,C 180,E1 -18770.444,E2 -18770.444} C_VEL
LIN {X 0,Y 281.566,Z 295.806,A -85,B 0,C 180,E1 -18770.685,E2 -18770.685} C_VEL
LIN {X 0,Y 276.361,Z 403.621,A -85,B 0,C 180,E1 -18773.472,E2 -18773.472} C_VEL
LIN {X 0,Y 274.747,Z 419.158,A -85,B 0,C 180,E1 -18774.132,E2 -18774.132} C_VEL
LIN {X 0,Y 272.687,Z 433.472,A -85,B 0,C 180,E1 -18775.01,E2 -18775.01} C_VEL
LIN {X 0,Y 270.115,Z 447.952,A -85,B 0,C 180,E1 -18776.212,E2 -18776.212} C_VEL
LIN {X 0,Y 267.566,Z 460.349,A -85,B 0,C 180,E1 -18777.528,E2 -18777.528} C_VEL
LIN {X 0,Y 264.375,Z 473.275,A -85,B 0,C 180,E1 -18779.222,E2 -18779.222} C_VEL
LIN {X 0,Y 261.057,Z 485.602,A -85,B 0,C 180,E1 -18781.236,E2 -18781.236} C_VEL
LIN {X 0,Y 258.22,Z 495.978,A -85,B 0,C 180,E1 -18783.316,E2 -18783.316} C_VEL
LIN {X 0,Y 255.136,Z 506.961,A -85,B 0,C 180,E1 -18786.028,E2 -18786.028} C_VEL
LIN {X 0,Y 252.809,Z 514.869,A -85,B 0,C 180,E1 -18788.387,E2 -18788.387} C_VEL
LIN {X 0,Y 250.659,Z 522.587,A -85,B 0,C 180,E1 -18791.19,E2 -18791.19} C_VEL
LIN {X 0,Y 248.856,Z 529.756,A -85,B 0,C 180,E1 -18794.438,E2 -18794.438} C_VEL
LIN {X 0,Y 247.667,Z 535.345,A -85,B 0,C 180,E1 -18797.713,E2 -18797.713} C_VEL
LIN {X 0,Y 247.203,Z 538.58,A -85,B 0,C 180,E1 -18800.179,E2 -18800.179} C_VEL
LIN {X 0,Y 247.016,Z 541.761,A -85,B 0,C 180,E1 -18803.466,E2 -18803.466} C_VEL
LIN {X 0,Y 247,Z 543.656,A -85,B 0,C 180,E1 -18806.738,E2 -18806.738} C_VEL
LIN {X 0,Y 247.09,Z 544.295,A -85,B 0,C 180,E1 -18810.001,E2 -18810.001} C_VEL
LIN {X 0,Y 247.013,Z 543.643,A -85,B 0,C 180,E1 -18813.263,E2 -18813.263} C_VEL
LIN {X 0,Y 247.018,Z 541.731,A -85,B 0,C 180,E1 -18816.535,E2 -18816.535} C_VEL
LIN {X 0,Y 247.209,Z 538.538,A -85,B 0,C 180,E1 -18819.822,E2 -18819.822} C_VEL
LIN {X 0,Y 247.954,Z 534.006,A -85,B 0,C 180,E1 -18823.106,E2 -18823.106} C_VEL
LIN {X 0,Y 249.42,Z 527.437,A -85,B 0,C 180,E1 -18826.66,E2 -18826.66} C_VEL
LIN {X 0,Y 251.505,Z 519.369,A -85,B 0,C 180,E1 -18830.018,E2 -18830.018} C_VEL
LIN {X 0,Y 253.986,Z 510.971,A -85,B 0,C 180,E1 -18832.793,E2 -18832.793} C_VEL
LIN {X 0,Y 256.905,Z 500.412,A -85,B 0,C 180,E1 -18835.625,E2 -18835.625} C_VEL
LIN {X 0,Y 259.705,Z 490.366,A -85,B 0,C 180,E1 -18837.828,E2 -18837.828} C_VEL
LIN {X 0,Y 262.845,Z 478.978,A -85,B 0,C 180,E1 -18839.868,E2 -18839.868} C_VEL
LIN {X 0,Y 266.004,Z 466.559,A -85,B 0,C 180,E1 -18841.676,E2 -18841.676} C_VEL
LIN {X 0,Y 268.658,Z 454.625,A -85,B 0,C 180,E1 -18843.087,E2 -18843.087} C_VEL
LIN {X 0,Y 271.138,Z 441.757,A -85,B 0,C 180,E1 -18844.317,E2 -18844.317} C_VEL
LIN {X 0,Y 273.389,Z 427.948,A -85,B 0,C 180,E1 -18845.339,E2 -18845.339} C_VEL
LIN {X 0,Y 275.311,Z 413.282,A -85,B 0,C 180,E1 -18846.123,E2 -18846.123} C_VEL
LIN {X 0,Y 276.436,Z 399.705,A -85,B 0,C 180,E1 -18846.631,E2 -18846.631} C_VEL
LIN {X 0,Y 281.495,Z 294.584,A -85,B 0,C 180,E1 -18849.324,E2 -18849.324} C_VEL
LIN {X 0,Y 280.766,Z 289.665,A -85,B 0,C 180,E1 -18849.602,E2 -18849.602} C_VEL
LIN {X 0,Y 273.776,Z 274.405,A -85,B 0,C 180,E1 -18851.282,E2 -18851.282} C_VEL
LIN {X 0,Y 266.507,Z 260.48,A -85,B 0,C 180,E1 -18853.102,E2 -18853.102} C_VEL
LIN {X 0,Y 259.603,Z 248.728,A -85,B 0,C 180,E1 -18854.919,E2 -18854.919} C_VEL
LIN {X 0,Y 257.333,Z 244.853,A -85,B 0,C 180,E1 -18855.607,E2 -18855.607} C_VEL
LIN {X 0,Y 254.261,Z 235.401,A -85,B 0,C 180,E1 -18859.492,E2 -18859.492} C_VEL
LIN {X 0,Y 251.536,Z 227.729,A -85,B 0,C 180,E1 -18863.079,E2 -18863.079} C_VEL
LIN {X 0,Y 249.052,Z 221.163,A -85,B 0,C 180,E1 -18866.615,E2 -18866.615} C_VEL
LIN {X 0,Y 249.092,Z 221.062,A -85,B 0,C 180,E1 -18871.338,E2 -18871.338} C_VEL
LIN {X 0,Y 249.151,Z 221.045,A -85,B 0,C 180,E1 -18874.969,E2 -18874.969} C_VEL
LIN {X 0,Y 249.111,Z 221.081,A -85,B 0,C 180,E1 -18880.212,E2 -18880.212} C_VEL
LIN {X 0,Y 249.242,Z 221.061,A -85,B 0,C 180,E1 -18883.622,E2 -18883.622} C_VEL
LIN {X 0,Y 249.244,Z 221.063,A -85,B 0,C 180,E1 -18888.616,E2 -18888.616} C_VEL
LIN {X 0,Y 249.454,Z 221.035,A -85,B 0,C 180,E1 -18891.902,E2 -18891.902} C_VEL
LIN {X 0,Y 249.295,Z 221.045,A -85,B 0,C 180,E1 -18895.149,E2 -18895.149} C_VEL
LIN {X 0,Y 249.675,Z 220.996,A -85,B 0,C 180,E1 -18898.387,E2 -18898.387} C_VEL
LIN {X 0,Y 249.675,Z 221.007,A -85,B 0,C 180,E1 -18901.613,E2 -18901.613} C_VEL
LIN {X 0,Y 249.45,Z 221.027,A -85,B 0,C 180,E1 -18906.755,E2 -18906.755} C_VEL
LIN {X 0,Y 249.389,Z 221.047,A -85,B 0,C 180,E1 -18909.735,E2 -18909.735} C_VEL
LIN {X 0,Y 249.202,Z 221.063,A -85,B 0,C 180,E1 -18914.704,E2 -18914.704} C_VEL
LIN {X 0,Y 249.14,Z 221.077,A -85,B 0,C 180,E1 -18918.078,E2 -18918.078} C_VEL
LIN {X 0,Y 249.105,Z 221.08,A -85,B 0,C 180,E1 -18921.517,E2 -18921.517} C_VEL
LIN {X 0,Y 249.131,Z 221.079,A -85,B 0,C 180,E1 -18925.482,E2 -18925.482} C_VEL
LIN {X 0,Y 249.074,Z 221.044,A -85,B 0,C 180,E1 -18928.989,E2 -18928.989} C_VEL
LIN {X 0,Y 249.037,Z 221.083,A -85,B 0,C 180,E1 -18932.425,E2 -18932.425} C_VEL
LIN {X 0,Y 249.099,Z 221.263,A -85,B 0,C 180,E1 -18935.985,E2 -18935.985} C_VEL
LIN {X 0,Y 251.046,Z 226.787,A -85,B 0,C 180,E1 -18939.041,E2 -18939.041} C_VEL
LIN {X 0,Y 253.633,Z 234.247,A -85,B 0,C 180,E1 -18942.756,E2 -18942.756} C_VEL
LIN {X 0,Y 256.468,Z 243.228,A -85,B 0,C 180,E1 -18946.759,E2 -18946.759} C_VEL
LIN {X 0,Y 257.021,Z 245.031,A -85,B 0,C 180,E1 -18947.345,E2 -18947.345} C_VEL
LIN {X 0,Y 263.178,Z 255.359,A -85,B 0,C 180,E1 -18949.016,E2 -18949.016} C_VEL
LIN {X 0,Y 270.015,Z 267.81,A -85,B 0,C 180,E1 -18950.745,E2 -18950.745} C_VEL
LIN {X 0,Y 277.158,Z 282.525,A -85,B 0,C 180,E1 -18952.472,E2 -18952.472} C_VEL
LIN {X 0,Y 279.474,Z 288.089,A -85,B 0,C 180,E1 -18953.029,E2 -18953.029} C_VEL
LIN {X 0,Y 280.966,Z 297.139,A -85,B 0,C 180,E1 -18953.544,E2 -18953.544} C_VEL
LIN {X 0,Y 277.03,Z 391.011,A -85,B 0,C 180,E1 -18955.8,E2 -18955.8} C_VEL
LIN {X 0,Y 275.774,Z 405.418,A -85,B 0,C 180,E1 -18956.393,E2 -18956.393} C_VEL
LIN {X 0,Y 273.991,Z 419.891,A -85,B 0,C 180,E1 -18957.298,E2 -18957.298} C_VEL
LIN {X 0,Y 271.721,Z 433.24,A -85,B 0,C 180,E1 -18958.415,E2 -18958.415} C_VEL
LIN {X 0,Y 269.229,Z 445.744,A -85,B 0,C 180,E1 -18959.775,E2 -18959.775} C_VEL
LIN {X 0,Y 266.448,Z 457.865,A -85,B 0,C 180,E1 -18961.44,E2 -18961.44} C_VEL
LIN {X 0,Y 263.697,Z 467.695,A -85,B 0,C 180,E1 -18963.058,E2 -18963.058} C_VEL
LIN {X 0,Y 260.551,Z 478.551,A -85,B 0,C 180,E1 -18965.286,E2 -18965.286} C_VEL
LIN {X 0,Y 257.6,Z 487.58,A -85,B 0,C 180,E1 -18967.545,E2 -18967.545} C_VEL
LIN {X 0,Y 255.283,Z 495.275,A -85,B 0,C 180,E1 -18969.926,E2 -18969.926} C_VEL
LIN {X 0,Y 253.154,Z 501.417,A -85,B 0,C 180,E1 -18972.219,E2 -18972.219} C_VEL
LIN {X 0,Y 251.309,Z 506.693,A -85,B 0,C 180,E1 -18974.593,E2 -18974.593} C_VEL
LIN {X 0,Y 249.536,Z 512.283,A -85,B 0,C 180,E1 -18977.805,E2 -18977.805} C_VEL
LIN {X 0,Y 248.624,Z 515.535,A -85,B 0,C 180,E1 -18980.235,E2 -18980.235} C_VEL
LIN {X 0,Y 247.759,Z 518.641,A -85,B 0,C 180,E1 -18983.484,E2 -18983.484} C_VEL
LIN {X 0,Y 247.315,Z 520.48,A -85,B 0,C 180,E1 -18986.741,E2 -18986.741} C_VEL
LIN {X 0,Y 247.108,Z 521.106,A -85,B 0,C 180,E1 -18989.999,E2 -18989.999} C_VEL
LIN {X 0,Y 247.297,Z 520.525,A -85,B 0,C 180,E1 -18993.258,E2 -18993.258} C_VEL
LIN {X 0,Y 247.713,Z 518.736,A -85,B 0,C 180,E1 -18996.516,E2 -18996.516} C_VEL
LIN {X 0,Y 248.541,Z 515.678,A -85,B 0,C 180,E1 -18999.767,E2 -18999.767} C_VEL
LIN {X 0,Y 249.879,Z 511.264,A -85,B 0,C 180,E1 -19003.002,E2 -19003.002} C_VEL
LIN {X 0,Y 251.754,Z 505.336,A -85,B 0,C 180,E1 -19006.209,E2 -19006.209} C_VEL
LIN {X 0,Y 254.144,Z 498.753,A -85,B 0,C 180,E1 -19008.96,E2 -19008.96} C_VEL
LIN {X 0,Y 256.656,Z 490.645,A -85,B 0,C 180,E1 -19011.693,E2 -19011.693} C_VEL
LIN {X 0,Y 259.393,Z 482.246,A -85,B 0,C 180,E1 -19013.979,E2 -19013.979} C_VEL
LIN {X 0,Y 262.51,Z 472.13,A -85,B 0,C 180,E1 -19016.214,E2 -19016.214} C_VEL
LIN {X 0,Y 265.637,Z 460.897,A -85,B 0,C 180,E1 -19018.223,E2 -19018.223} C_VEL
LIN {X 0,Y 268.758,Z 448.419,A -85,B 0,C 180,E1 -19020.004,E2 -19020.004} C_VEL
LIN {X 0,Y 271.261,Z 436.08,A -85,B 0,C 180,E1 -19021.426,E2 -19021.426} C_VEL
LIN {X 0,Y 273.629,Z 422.399,A -85,B 0,C 180,E1 -19022.64,E2 -19022.64} C_VEL
LIN {X 0,Y 275.583,Z 408.042,A -85,B 0,C 180,E1 -19023.577,E2 -19023.577} C_VEL
LIN {X 0,Y 276.887,Z 393.895,A -85,B 0,C 180,E1 -19024.219,E2 -19024.219} C_VEL
LIN {X 0,Y 277.99,Z 372.605,A -85,B 0,C 180,E1 -19024.778,E2 -19024.778} C_VEL
LIN {X 0,Y 281.034,Z 297.042,A -85,B 0,C 180,E1 -19026.582,E2 -19026.582} C_VEL
LIN {X 0,Y 279.2,Z 287.036,A -85,B 0,C 180,E1 -19027.185,E2 -19027.185} C_VEL
LIN {X 0,Y 272.139,Z 271.946,A -85,B 0,C 180,E1 -19028.873,E2 -19028.873} C_VEL
LIN {X 0,Y 266.469,Z 261.124,A -85,B 0,C 180,E1 -19030.285,E2 -19030.285} C_VEL
LIN {X 0,Y 259.092,Z 248.407,A -85,B 0,C 180,E1 -19032.22,E2 -19032.22} C_VEL
LIN {X 0,Y 256.82,Z 244.404,A -85,B 0,C 180,E1 -19032.938,E2 -19032.938} C_VEL
LIN {X 0,Y 254.048,Z 235.559,A -85,B 0,C 180,E1 -19036.789,E2 -19036.789} C_VEL
LIN {X 0,Y 251.788,Z 228.84,A -85,B 0,C 180,E1 -19040.06,E2 -19040.06} C_VEL
LIN {X 0,Y 249.7,Z 223.222,A -85,B 0,C 180,E1 -19043.091,E2 -19043.091} C_VEL
LIN {X 0,Y 249.078,Z 221.139,A -85,B 0,C 180,E1 -19044.36,E2 -19044.36} C_VEL
LIN {X 0,Y 249.037,Z 221.086,A -85,B 0,C 180,E1 -19047.844,E2 -19047.844} C_VEL
LIN {X 0,Y 249.082,Z 221.043,A -85,B 0,C 180,E1 -19051.336,E2 -19051.336} C_VEL
LIN {X 0,Y 249.148,Z 221.074,A -85,B 0,C 180,E1 -19054.968,E2 -19054.968} C_VEL
LIN {X 0,Y 249.123,Z 221.077,A -85,B 0,C 180,E1 -19058.582,E2 -19058.582} C_VEL
LIN {X 0,Y 249.238,Z 221.052,A -85,B 0,C 180,E1 -19063.621,E2 -19063.621} C_VEL
LIN {X 0,Y 249.248,Z 221.05,A -85,B 0,C 180,E1 -19068.616,E2 -19068.616} C_VEL
LIN {X 0,Y 249.257,Z 221.05,A -85,B 0,C 180,E1 -19068.923,E2 -19068.923} C_VEL
LIN {X 0,Y 248.624,Z 221.142,A -85,B 0,C 180,E1 -19070.274,E2 -19070.274} C_VEL
LIN {X 0,Y 245.751,Z 221.496,A -85,B 0,C 180,E1 -19072.477,E2 -19072.477} C_VEL
LIN {X 0,Y 243.33,Z 221.799,A -85,B 0,C 180,E1 -19074.271,E2 -19074.271} C_VEL
LIN {X 0,Y 242.354,Z 221.914,A -85,B 0,C 180,E1 -19075.664,E2 -19075.664} C_VEL
LIN {X 0,Y 242.31,Z 221.914,A -85,B 0,C 180,E1 -19076.135,E2 -19076.135} C_VEL
LIN {X 0,Y 242.631,Z 221.883,A -85,B 0,C 180,E1 -19078.34,E2 -19078.34} C_VEL
LIN {X 0,Y 242.631,Z 221.873,A -85,B 0,C 180,E1 -19081.66,E2 -19081.66} C_VEL
LIN {X 0,Y 242.428,Z 221.904,A -85,B 0,C 180,E1 -19086.659,E2 -19086.659} C_VEL
LIN {X 0,Y 242.309,Z 221.914,A -85,B 0,C 180,E1 -19090.022,E2 -19090.022} C_VEL
LIN {X 0,Y 242.161,Z 221.939,A -85,B 0,C 180,E1 -19095.141,E2 -19095.141} C_VEL
LIN {X 0,Y 242.068,Z 221.948,A -85,B 0,C 180,E1 -19098.624,E2 -19098.624} C_VEL
LIN {X 0,Y 242.008,Z 221.956,A -85,B 0,C 180,E1 -19102.18,E2 -19102.18} C_VEL
LIN {X 0,Y 242.062,Z 221.919,A -85,B 0,C 180,E1 -19105.838,E2 -19105.838} C_VEL
LIN {X 0,Y 242.011,Z 221.949,A -85,B 0,C 180,E1 -19110.544,E2 -19110.544} C_VEL
LIN {X 0,Y 242.047,Z 222.276,A -85,B 0,C 180,E1 -19111.388,E2 -19111.388} C_VEL
LIN {X 0,Y 244.503,Z 228.685,A -85,B 0,C 180,E1 -19115.091,E2 -19115.091} C_VEL
LIN {X 0,Y 246.446,Z 233.978,A -85,B 0,C 180,E1 -19117.815,E2 -19117.815} C_VEL
LIN {X 0,Y 249.192,Z 241.953,A -85,B 0,C 180,E1 -19121.511,E2 -19121.511} C_VEL
LIN {X 0,Y 250.299,Z 245.19,A -85,B 0,C 180,E1 -19122.788,E2 -19122.788} C_VEL
LIN {X 0,Y 259.12,Z 259.692,A -85,B 0,C 180,E1 -19125.338,E2 -19125.338} C_VEL
LIN {X 0,Y 265.955,Z 272.247,A -85,B 0,C 180,E1 -19127.164,E2 -19127.164} C_VEL
